	MW(WORD_STRONG :=  MesBlock3_Temp[1  ],	WORD_WEAK := MesBlock3_Temp[2  ], SIZE := 2, FIX := 3, SIGNED := 1, VAR_OUT	:= MesDataExd.MesData.MesIdc);
	MW(WORD_STRONG :=  MesBlock3_Temp[3  ],	WORD_WEAK := MesBlock3_Temp[4  ], SIZE := 2, FIX := 2, SIGNED := 1, VAR_OUT	:= MesDataExd.MesData.MesUdc);
	MW(WORD_STRONG :=  MesBlock3_Temp[5  ],	WORD_WEAK := MesBlock3_Temp[6  ], SIZE := 2, FIX := 0, SIGNED := 1, VAR_OUT	:= MesDataExd.MesData.MesPdc);
	MW(WORD_STRONG :=  MesBlock3_Temp[7  ],	WORD_WEAK := MesBlock3_Temp[8  ], SIZE := 2, FIX := 0, SIGNED := 1, VAR_OUT	:= MesDataExd.MesData.MesP);
	MW(WORD_STRONG :=  MesBlock3_Temp[21 ],	WORD_WEAK := MesBlock3_Temp[22 ], SIZE := 2, FIX := 2, SIGNED := 0, VAR_OUT	:= MesDataExd.MesU12);
	MW(WORD_STRONG :=  MesBlock3_Temp[23 ],	WORD_WEAK := MesBlock3_Temp[24 ], SIZE := 2, FIX := 2, SIGNED := 0, VAR_OUT	:= MesDataExd.MesU23);
	MW(WORD_STRONG :=  MesBlock3_Temp[25 ],	WORD_WEAK := MesBlock3_Temp[26 ], SIZE := 2, FIX := 2, SIGNED := 0, VAR_OUT	:= MesDataExd.MesU31);
	MW(WORD_STRONG :=  MesBlock3_Temp[27 ],	WORD_WEAK := MesBlock3_Temp[28 ], SIZE := 2, FIX := 3, SIGNED := 0, VAR_OUT	:= MesDataExd.MesData.MesI);
	MW(WORD_STRONG :=  MesBlock3_Temp[29 ],	WORD_WEAK := MesBlock3_Temp[30 ], SIZE := 2, FIX := 3, SIGNED := 0, VAR_OUT	:= MesDataExd.MesI1);
	MW(WORD_STRONG :=  MesBlock3_Temp[31 ],	WORD_WEAK := MesBlock3_Temp[32 ], SIZE := 2, FIX := 3, SIGNED := 0, VAR_OUT	:= MesDataExd.MesI2);
	MW(WORD_STRONG :=  MesBlock3_Temp[33 ],	WORD_WEAK := MesBlock3_Temp[34 ], SIZE := 2, FIX := 3, SIGNED := 0, VAR_OUT	:= MesDataExd.MesI3);
	MW(WORD_STRONG :=  MesBlock3_Temp[35 ],	WORD_WEAK := MesBlock3_Temp[36 ], SIZE := 2, FIX := 2, SIGNED := 0, VAR_OUT	:= MesDataExd.MesData.MesFreq);
	MW(WORD_STRONG :=  MesBlock3_Temp[37 ],	WORD_WEAK := MesBlock3_Temp[38 ], SIZE := 2, FIX := 2, SIGNED := 1, VAR_OUT	:= MesDataExd.MesData.MesQ);
	MW(WORD_STRONG :=  MesBlock3_Temp[53 ],	WORD_WEAK := MesBlock3_Temp[54 ], SIZE := 2, FIX := 2, SIGNED := 0, VAR_OUT	:= MesDataExd.MesData.MesCosPhi);
	MW(WORD_STRONG :=  MesBlock3_Temp[55 ],	WORD_WEAK := MesBlock3_Temp[56 ], SIZE := 2, FIX := 0, SIGNED := 0, VAR_OUT	:= MesDataExd.MesTypeCosPhi);
	MW(WORD_STRONG :=  MesBlock3_Temp[57 ],	WORD_WEAK := MesBlock3_Temp[58 ], SIZE := 2, FIX := 0, SIGNED := 0, VAR_OUT	:= MesDataExd.MesQMode);
	MW(WORD_STRONG :=  MesBlock3_Temp[59 ],	WORD_WEAK := MesBlock3_Temp[60 ], SIZE := 2, FIX := 0, SIGNED := 1, VAR_OUT	:= MesDataExd.MesSetptQ);
	MW(WORD_STRONG :=  MesBlock3_Temp[61 ],	WORD_WEAK := MesBlock3_Temp[62 ], SIZE := 2, FIX := 1, SIGNED := 1, VAR_OUT	:= MesDataExd.MesSetptQ_Pct);
	MW(WORD_STRONG :=  MesBlock3_Temp[63 ],	WORD_WEAK := MesBlock3_Temp[64 ], SIZE := 2, FIX := 2, SIGNED := 1, VAR_OUT	:= MesDataExd.MesSetptCosPhi);
	MW(WORD_STRONG :=  MesBlock3_Temp[65 ],	WORD_WEAK := MesBlock3_Temp[66 ], SIZE := 2, FIX := 0, SIGNED := 0, VAR_OUT	:= MesDataExd.MesSetptType_CosPhi);
	MW(WORD_STRONG :=  MesBlock3_Temp[67 ],	WORD_WEAK := MesBlock3_Temp[68 ], SIZE := 2, FIX := 0, SIGNED := 0, VAR_OUT	:= MesDataExd.MesPMode);
	MW(WORD_STRONG :=  MesBlock3_Temp[69 ],	WORD_WEAK := MesBlock3_Temp[70 ], SIZE := 2, FIX := 0, SIGNED := 0, VAR_OUT	:= MesDataExd.MesPSetpt);
	MW(WORD_STRONG :=  MesBlock3_Temp[71 ],	WORD_WEAK := MesBlock3_Temp[72 ], SIZE := 2, FIX := 0, SIGNED := 0, VAR_OUT	:= MesDataExd.MesPSetptPct);
	MW(WORD_STRONG :=  MesBlock3_Temp[73 ],	WORD_WEAK := MesBlock3_Temp[74 ], SIZE := 2, FIX := 2, SIGNED := 0, VAR_OUT	:= MesDataExd.MesData.MesV);
	
	MW(WORD_STRONG :=  MesBlock4_Temp[1  ],	WORD_WEAK := MesBlock4_Temp[2  ], SIZE := 2, FIX := 1, SIGNED := 1, VAR_OUT	:= MesDataExd.MesTmpHs);
	MW(WORD_STRONG :=  MesBlock4_Temp[5  ],	WORD_WEAK := MesBlock4_Temp[6  ], SIZE := 2, FIX := 1, SIGNED := 1, VAR_OUT	:= MesDataExd.MesTmpCab1);
	MW(WORD_STRONG :=  MesBlock4_Temp[9  ],	WORD_WEAK := MesBlock4_Temp[10 ], SIZE := 2, FIX := 1, SIGNED := 1, VAR_OUT	:= MesDataExd.MesTmpCab3);
	MW(WORD_STRONG :=  MesBlock4_Temp[17 ],	WORD_WEAK := MesBlock4_Temp[18 ], SIZE := 2, FIX := 1, SIGNED := 1, VAR_OUT	:= MesDataExd.MesTmpExt);
	MW(WORD_STRONG :=  MesBlock4_Temp[37 ],	WORD_WEAK := MesBlock4_Temp[38 ], SIZE := 2, FIX := 1, SIGNED := 1, VAR_OUT	:= MesDataExd.MesTmpCol);
			                                                                                                                          

	MW(WORD_STRONG :=  MesBlock5_Temp[1  ],	WORD_WEAK := MesBlock5_Temp[2  ], SIZE := 2, FIX := 0, SIGNED := 0, VAR_OUT	:= MesDataExd.MesGHI);
	MW(WORD_STRONG :=  MesBlock5_Temp[25 ],	WORD_WEAK := MesBlock5_Temp[26 ], SIZE := 2, FIX := 0, SIGNED := 0, VAR_OUT	:= MesDataExd.MesInCur1);
	MW(WORD_STRONG :=  MesBlock5_Temp[27 ],	WORD_WEAK := MesBlock5_Temp[28 ], SIZE := 2, FIX := 0, SIGNED := 0, VAR_OUT	:= MesDataExd.MesInCur2);

	
	MW(WORD_STRONG :=  MesBlock6_Temp[1  ],	WORD_WEAK := MesBlock6_Temp[2  ], SIZE := 2, FIX := 0, SIGNED := 0, VAR_OUT	:= PosInterm);
	MesDataExd.MesOpStateOn := SEL(PosInterm = 381,SEL(PosInterm=569,FALSE, TRUE), FALSE);
	MW(WORD_STRONG :=  MesBlock6_Temp[12 ],	WORD_WEAK := MesBlock6_Temp[13 ], SIZE := 2, FIX := 0, SIGNED := 0, VAR_OUT	:= PosInterm);
	MesDataExd.MesbRIsoOn := SEL(PosInterm=303,SEL(PosInterm=308,FALSE, TRUE), FALSE);
	IdcTotal := 0;


	IF FB_ModbusRead[7].OUT_NbRead > 0 THEN 
		
		MW(WORD_STRONG :=  MesBlock7_Temp[1 ],	WORD_WEAK := MesBlock7_Temp[2], SIZE := 2, FIX := 3, SIGNED := 1, VAR_OUT	:= MesDataExd.BJMonitor[ID_SSM].AX_STR[1].MesData.MesIdc);
		MW(WORD_STRONG :=  MesBlock7_Temp[3 ],	WORD_WEAK := MesBlock7_Temp[4], SIZE := 2, FIX := 3, SIGNED := 1, VAR_OUT	:= MesDataExd.BJMonitor[ID_SSM].AX_STR[2].MesData.MesIdc);
		MW(WORD_STRONG :=  MesBlock7_Temp[5 ],	WORD_WEAK := MesBlock7_Temp[6 ], SIZE := 2, FIX := 3, SIGNED := 1, VAR_OUT	:= MesDataExd.BJMonitor[ID_SSM].AX_STR[3].MesData.MesIdc);
		MW(WORD_STRONG :=  MesBlock7_Temp[7 ],	WORD_WEAK := MesBlock7_Temp[8 ], SIZE := 2, FIX := 3, SIGNED := 1, VAR_OUT	:= MesDataExd.BJMonitor[ID_SSM].AX_STR[4].MesData.MesIdc);
		MW(WORD_STRONG :=  MesBlock7_Temp[9 ],	WORD_WEAK := MesBlock7_Temp[10], SIZE := 2, FIX := 3, SIGNED := 1, VAR_OUT	:= MesDataExd.BJMonitor[ID_SSM].AX_STR[5].MesData.MesIdc);
		MW(WORD_STRONG :=  MesBlock7_Temp[11],	WORD_WEAK := MesBlock7_Temp[12], SIZE := 2, FIX := 3, SIGNED := 1, VAR_OUT	:= MesDataExd.BJMonitor[ID_SSM].AX_STR[6].MesData.MesIdc);
		MW(WORD_STRONG :=  MesBlock7_Temp[13],	WORD_WEAK := MesBlock7_Temp[14], SIZE := 2, FIX := 3, SIGNED := 1, VAR_OUT	:= MesDataExd.BJMonitor[ID_SSM].AX_STR[7].MesData.MesIdc);
		MW(WORD_STRONG :=  MesBlock7_Temp[15],	WORD_WEAK := MesBlock7_Temp[16], SIZE := 2, FIX := 3, SIGNED := 1, VAR_OUT	:= MesDataExd.BJMonitor[ID_SSM].AX_STR[8].MesData.MesIdc);	
	
			
		//	MW(WORD_STRONG :=  MesBlock8_Temp[1],	WORD_WEAK := MesBlock8_Temp[2 ], SIZE := 2, FIX := 2, SIGNED := 0, VAR_OUT	:= PosInterm);
		//MesDataExd.BJMonitor.MesID_SignalContact1 := SEL(PosInterm=303,SEL(PosInterm=308,FALSE, TRUE), FALSE);
		MesDataExd.BJMonitor[ID_SSM].MesID_SignalContact1 := MesBlock8_Temp[1] ; 
		//	MW(WORD_STRONG :=  MesBlock8_Temp[3],	WORD_WEAK := MesBlock8_Temp[4 ], SIZE := 2, FIX := 2, SIGNED := 0, VAR_OUT	:= PosInterm);
		//MesDataExd.BJMonitor.MesID_SignalContact2 := SEL(PosInterm=303,SEL(PosInterm=308,FALSE, TRUE), FALSE);
		MesDataExd.BJMonitor[ID_SSM].MesID_SignalContact2 := MesBlock8_Temp[3] ; 
			

		ID_SSM := ID_SSM +1 MOD 7 ; 
		IF ID_SSM = 0 THEN 
			ID_SSM := 1 ; 
		END_IF
	END_IF




	MesDataExd.MesData.MesP := MesDataExd.MesData.MesP/1000;
	MesDataExd.MesData.MesPdc := MesDataExd.MesData.MesPdc/1000;
	MesDataExd.MesData.MesQ := MesDataExd.MesData.MesQ/1000;
	MesDataExd.MesPSetpt := MesDataExd.MesPSetpt / 1000;
	MesDataExd.MesSetptQ := MesDataExd.MesSetptQ / 1000;

	
	
END_IF
	
	
// Update value 
MesDataExd.Mesdata.ParamPn		:= ParamPn ; 
MesDataExd.Mesdata.ParamQn		:= ParamQn ; 
	


FOR KK := 1 TO CstNbSB_INV_G DO 
	MesDataExd.BJMonitor[KK].MesClosed_DCSwitch := IN_MesClosed_BJ_IO[KK] ; 
END_FOR
END_METHOD

METHOD M_StartStop 
VAR_INPUT
END_VAR
VAR
	KK : UINT;
	AX_ADR_MB			: WORD := 40009;
	AX_QTY_MB			: ARRAY[1..2] OF BYTE := [2, 2];
	MotStart			: WORD := 569;
	MotStop				: WORD := 381;
	
END_VAR
SUPER^.M_StartStop() ; 
FB_ModbusWrite[3](WriteCmd := FALSE);

//Read the setpoints
	// Evaluate the cmd given 

	StartStop_RTrig(CLK:=CalCP_CMD_StartStop);
	StartStop_RTrigIO(CLK:=CalCP_CMD_StartStopIO);
	
//	IF StartStop_RTrig.Q THEN
		IF RS_StartStop.Q1 THEN
			MesBlockWrite3_Temp[1] := 0;
			MesBlockWrite3_Temp[2] := MotStart;
		ELSE 
			MesBlockWrite3_Temp[1] := 0;
			MesBlockWrite3_Temp[2] := MotStop;
		END_IF
//	END_IF
	
//	IF StartStop_RTrigIO.Q THEN
//		IF Cmd_SwitchOff THEN
//			Cmd_SwitchOff		:= 0;
//		ELSIF NOT Cmd_SwitchOff THEN
//			Cmd_SwitchOff		:= 1;
//		END_IF
//	END_IF
OUT_Cmd_SwitchOff_IO	:= CalCP_CMD_StartStopIO	;
	

MesDataExd.Mesdata.OUT_CmdStart := RS_StartStop.Q1 ;
MesDataExd.Mesdata.OUT_CmdStop := NOT RS_StartStop.Q1 ;

	
	FB_ModbusWrite[3]
	(
		pSrcAddr := ADR (MesBlockWrite3_Temp),
		sIPAddr := ParamIPAddress,
		tTimeout := ParamTimeout,
		nMBAddr := AX_ADR_MB,
		nTCPport := ParamTCPPort,
		cbLength := SIZEOF(MesBlockWrite3_Temp),
		nQuantity := 2,
		nUnitID := 3,
		WriteCmd := CalCP_CMD_StartStop AND MesDataExd.mesData.MesCP_Write ,
		Reset := CmdClearFault_G,
		ErrorId => AX_ModbusWriteAlarmId[3],
		ModbusWriteAlarm => AX_ModbusWriteAlarm[3]
	);


SUPER^.M_Curtail() ;
END_METHOD

METHOD M_StateManager
//////////////////
// Detect which is the state of the inverter. IF loss of communication MesState =0 , the last inverter state is kept .  
/////////////////

VAR 
	// Method local variables (reinitialized at each cycle) 

	
END_VAR
// 0 = Stopped, 1 = MPPT, 2 = Sleeping, 3 = Starting, 4 = Throttled, 5 = Shutting down, 6 = Fault, 7 = Standby

MesDataExd.Mesdata.MesState 			:= 0  ; 

IF MesDataExd.mesData.MesState_Inv = 381 OR MesDataExd.mesData.MesState_Inv = 1455 THEN // IF INVERTER IS STOPPED 309 = Operation && 455 = warning
	MesDataExd.Mesdata.MesState.0 := 1;		// Stop
ELSIF MesDataExd.mesData.MesState_Inv = 295 THEN
	MesDataExd.Mesdata.MesState.1 := 1;
ELSIF MesDataExd.mesData.MesState_Inv = 1466 THEN // Wait 
	MesDataExd.Mesdata.MesState.7 := 1;
ELSIF MesDataExd.mesData.MesState_Inv = 1467 OR MesDataExd.mesData.MesState_Inv = 1468 OR MesDataExd.mesData.MesState_Inv = 1479 THEN
	MesDataExd.Mesdata.MesState.3 := 1;
ELSIF MesDataExd.mesData.MesState_Inv = 1469  THEN
	MesDataExd.Mesdata.MesState.5 := 1;
ELSIF MesDataExd.mesData.MesState_Inv = 1470  THEN
	MesDataExd.Mesdata.MesState.6 := 1;
ELSE 
	MesDataExd.Mesdata.MesState.0 := 1;
END_IF

//IF MesDataExd.Mesdata.OUT_SetptP < ParamPn AND MesDataExd.Mesdata.MesP > 0.95 * MesDataExd.Mesdata.OUT_SetptP THEN
//	MesDataExd.Mesdata.MesIDState.4 := 1;
//END_IF



SUPER^.M_StateManager() ;
END_METHOD

END_FUNCTION_BLOCK

// ---- 01_Equipement_Library/Inverter/FB_INV_SmaSCXXXXUP_US.TcPOU
FUNCTION_BLOCK FB_INV_SmaSCXXXXUP_US EXTENDS FB_INV_Base
// Reading through Webbox . Curtailement not possible through modbus . 
//

VAR_INPUT PERSISTENT
	ParamTcpPort				: UINT	:= 502 ;	(* Modbus TCP port*)
	//{attribute 'OPC.UA.DA' := '1'} 
	//ParamQn						: REAL ;		(* (kVAr) Nominal Reactive Power*)
	{attribute 'OPC.UA.DA' := '1'} 
	ParamIPAddress				: STRING; 			(* (NA)Config: IP Adress of PV INverter	*)
	{attribute 'OPC.UA.DA' := '1'} 
	ParamUnitID 				: BYTE := 3; 			(* (NA)   SMA Modbus Unit ID. *)
	ParamNumInv					: BYTE;             (* Inverter Index  *)
	ParamNbSB					: BYTE :=5 ; (* Number of String Box per inverter*)
	ParamNbSTR					: BYTE :=8 ; (* Number of String per string Box*)
	
//	ParamUnitID_STR				: ARRAY[1..CstNbSB_INV_G] OF BYTE ; (* Unit ID Arrray for each string box . *)
	
	ParamDelayReadSTR			: TIME := T#2S ; 			(* (s) Delay after inv data read , to read string values . 	*)

END_VAR

VAR_INPUT 
	// Parameters of the Object (instance specific) 
	       	MesDataExd					: INV_SmaSCXXXXUP_US;
	                                     	
END_VAR

VAR
		
	// M_ALARMMNGMT VARIABLES //
	
	// M_READ VARIABLES//
		//MesDataCC_Read				:  INV_CC;	
		//MesDataCC_Cmd				:  INV_CC;
		
	
		FB_ModbusRead	          	: ARRAY[1..6] OF FB_ModbusReadInputRegs; 	            // (NA) FB for Modbus Reading
		FB_ModbusWrite				: ARRAY[1..3] OF FB_ModbusWrite;
		AX_ModbusReadAlarm			: ARRAY[1..6] OF BOOL;
		AX_ModbusReadAlarmId		: ARRAY[1..6] OF UDINT;		
		AX_ModbusWriteAlarm			: ARRAY[1..2] OF BOOL;
		AX_ModbusWriteAlarmId		: ARRAY[1..2] OF UDINT;
	

		
		MesBlock_Temp_1 				: ARRAY [1..125] OF WORD ; 		// (NA) Temporary Block with multiple modbus reading (Caution : Double Word variables)
		MesBlock_Temp_2 				: ARRAY [1..125] OF WORD ; 		// (NA) Temporary Block with multiple modbus reading (Caution : Double Word variables)
		MesBlock_Temp_3 				: ARRAY [1..125] OF WORD ; 		// (NA) Temporary Block with multiple modbus reading (Caution : Double Word variables)
		MesBlock_Temp_4 				: ARRAY [1..20] OF WORD ; 		// (NA) Temporary Block with multiple modbus reading (Caution : Double Word variables)
		MesBlock_Temp_5 				: ARRAY [1..20] OF WORD ; 		// (NA) Temporary Block with multiple modbus reading (Caution : Double Word variables)
		MesBlock_Temp_6				: ARRAY [1..20] OF WORD ;		// (NA) Temporary block with both start commands for each inverter


		MesBlockWrite3_Temp			: ARRAY [1..2] OF WORD ;
		
		TON_ReadSTR					: TON ; // Manage time delay fro reading string values. 
		
	// M_STARTSTOP//
	
		
	
	//  CUrtail 
	
		InvSetptP_temp		: WORD;
		InvSetptQ_temp		: WORD;
		
		MesBlockWrite1_Temp : WORD ; 
		MesBlockWrite2_Temp : WORD ; 
		
		
	// M_CP
		CalCP_CMD_StartStop			: BOOL ; 		  // Write command start;
	
	// M_STATEMANAGER//
	
	//M_EXECUTE VARIABLES //
	//	bInit						: BOOL ;
	//EMULATOR VARIABLES //
		
END_VAR

METHOD M_AlarmManagement
//////////////////
// Manages IntelliGen Alarms
/////////////////

VAR 
	// Method local variables (reinitialized at each cycle) 
	FB_AlarmCodeManager : FB_AlarmCodeManager ; 
	KK				: BYTE;		// For Loop 
	bComError		: BOOL := TRUE;
	bComWarning 	: BOOL;

END_VAR
FOR KK := 1 TO 4 DO
	bCOmError := bCOmError AND FB_ModbusRead[KK].ModbusReadAlarm;
	bComWarning := bComWarning OR FB_ModbusRead[KK].ModbusReadAlarm;
END_FOR
bComError := bComError AND FB_ModbusWrite[1].ModbusWriteAlarm ;
bComWarning := bComError OR FB_ModbusWrite[1].ModbusWriteAlarm  ;

TON_ComAlarm(IN := bComError, PT := T#30S , Q=> MesDataExd.MesData.MesAlarmCom);
TON_ComWarning(IN := bComWarning, PT := T#30S);



// ALARM CODE //
	FB_AlarmCodeManager(
		bAlarm1			:= MesDataExd.MesData.MesState_Inv  = 1392	, 	//Inverter in error  #Equipment
		bAlarm2			:= MesDataExd.MesData.MesState_Inv = 381,		// INV in stopped mode  #Equipment
		bAlarm3			:= MesDataExd.MesID_ErrorState = 1392 , 		// INV error synthesis #Equipment 
		bAlarm4			:= MesDataExd.Mesdata.MesOpened_Ac , 			// AC Switch is opened #Equipment
		bAlarm5			:= MesDataExd.Mesdata.MesOpened_Dc, 			// All DC switch are opened 
		bAlarm6			:= FALSE , //
		bAlarm7			:= FALSE , //
		bAlarm8			:= FALSE,						// 
		bAlarm9			:= FALSE	,					//
		bAlarm10		:= FALSE , 							// 
		bAlarm11		:= FALSE,								// 
		bAlarm12		:= FALSE,								// 
		bAlarm13		:= FALSE,  								//
		bAlarm14		:= FALSE,								// 
		bAlarm15		:= MesDataExd.MesData.MesAlarmCom, 						// No communication frames for the past 30 seconds #COM
		wAlarmCode		=> mesdataExd.MesData.MesAlarmCode);

// WARNING CODE //
	FB_AlarmCodeManager(
 		bAlarm1			:= FALSE, 													// 
		bAlarm2			:= FALSE,
		bAlarm3			:= NOT MesDataExd.MesData.MesCP_Read, 	  							// Reading has been disabled
		bAlarm4			:= FALSE,															// 
		bAlarm5			:= NOT MesDataExd.MesData.MesCP_Write,								// Writing has been disabled			
		bAlarm6			:= MesDataExd.MesID_DC1State = 311 OR MesDataExd.MesID_DC2State = 311 OR MesDataExd.MesID_DC3State = 311, // At least one DC switch is opened 								// 
		bAlarm7			:= FALSE , //
		bAlarm8			:= FALSE, 															//
		bAlarm9			:= FALSE, 								// 
		bAlarm10		:= NOT RS_StartStop_Local.Q1,                  						// Local Stop Command, 
		bAlarm11		:= FALSE, //
		bAlarm12		:= FALSE, //
		bAlarm13		:= FALSE, //
		bAlarm14		:= FALSE, //
		bAlarm15		:= TON_ComWarning.Q, 												//One or more than error, communication frames for the past 30 seconds #COM
		wAlarmCode		=> MesDataExd.mesdata.MesWarningCode);	

// EVENT CODE //
	FB_AlarmCodeManager(
		bAlarm1			:= MesDataExd.MesData.MesState_Inv = 1787, 								// Inverter status : Init  #Equipment
		bAlarm2			:= MesDataExd.MesData.MesState_Inv = 3522,								// Inverter status : Update  #Equipment
		bAlarm3			:= MesDataExd.MesData.MesState_Inv = 3523,								// Inverter status : Reset  #Equipment
		bAlarm4			:= MesDataExd.MesData.MesState_Inv = 1394,								// Inverter status : WaitAC  #Equipment
		bAlarm5			:= MesDataExd.MesData.MesState_Inv = 3524,								// Inverter status : ConnectAC  #Equipment
		bAlarm6			:= MesDataExd.MesData.MesState_Inv = 1393,								// Inverter status : WaitDC  #Equipment
		bAlarm7			:= NOT RS_StartStop.Q1, 				// Stop command for INV1
		bAlarm8			:= MesDataExd.MesData.MesState_Inv = 3525,								// Inverter status : ConnectDC  #Equipment
		bAlarm9			:= MesDataExd.MesData.MesState_Inv = 3526,								// Inverter status : GridFeed  #Equipment
		bAlarm10		:= MesDataExd.MesData.MesState_Inv = 3527,								// Inverter status : FRT  #Equipment
		bAlarm11		:= MesDataExd.MesData.MesState_Inv = 3528,								// Inverter status : Standby  #Equipment
		bAlarm12		:= MesDataExd.MesData.MesState_Inv = 3529,								// Inverter status : QonDemand  #Equipment
		bAlarm13		:= MesDataExd.MesData.MesState_Inv = 3530,								// Inverter status : RampDown   #Equipment
		bAlarm14		:= MesDataExd.MesData.MesState_Inv = 1469,								// Inverter status : ShutDown  #Equipment
		bAlarm15		:= MesDataExd.MesData.MesState_Inv = 375,								// Inverter status : Selftest  #Equipment
		wAlarmCode		=> mesdataExd.MesData.MesEventCode);

FB_AlarmCodeManager(
		bAlarm1			:= MesDataExd.MesID_Derating = 21585, 								// Inverter Derating : Stk.DcAmpLim  #Equipment
		bAlarm2			:= MesDataExd.MesID_Derating = 21586,								// Inverter Derating : Frt  #Equipment
		bAlarm3			:= MesDataExd.MesID_Derating = 21587,								// Inverter Derating : AmpGra  #Equipment
		bAlarm4			:= MesDataExd.MesID_Derating = 21588,								// Inverter Derating : AMax  #Equipment
		bAlarm5			:= MesDataExd.MesID_Derating = 21589,								// Inverter Derating : VAMax  #Equipment
		bAlarm6			:= MesDataExd.MesID_Derating = 21590,								// Inverter Derating : WCtlLoHz  #Equipment
		bAlarm7			:= MesDataExd.MesID_Derating = 21591,								// Inverter Derating : WCtlHz  #Equipment
		bAlarm8			:= MesDataExd.MesID_Derating = 21592,								// Inverter Derating : WGraRecon  #Equipment
		bAlarm9			:= MesDataExd.MesID_Derating = 21593,								// Inverter Derating : WGra  #Equipment
		bAlarm10		:= MesDataExd.MesID_Derating = 21594,								// Inverter Derating : WMax  #Equipment
		bAlarm11		:= MesDataExd.MesID_Derating = 21595,								// Inverter Derating : WMaxExt  #Equipment
		bAlarm12		:= MesDataExd.MesID_Derating = 21596,								// Inverter Derating : VecLen  #Equipment
		bAlarm13		:= MesDataExd.MesID_Derating = 21599,								// Inverter Derating : WGraStr   #Equipment
		bAlarm14		:= MesDataExd.MesID_Derating = 21601,								// Inverter Derating : WCtlVol  #Equipment
		bAlarm15		:= MesDataExd.MesID_Derating = 21602,								// Inverter Derating : Mvps.WRvLim  #Equipment
		wAlarmCode		=> mesdataExd.MesStatus_Derating);

FB_AlarmCodeManager(
		bAlarm1			:= MesDataExd.MesID_Derating = 21651, 								// Inverter Derating : VArPrio  #Equipment
		bAlarm2			:= FALSE,
		bAlarm3			:= FALSE,
		bAlarm4			:= FALSE,
		bAlarm5			:= FALSE,
		bAlarm6			:= FALSE,
		bAlarm7			:= FALSE,
		bAlarm8			:= FALSE,
		bAlarm9			:= FALSE,
		bAlarm10		:= FALSE,
		bAlarm11		:= FALSE,
		bAlarm12		:= FALSE,
		bAlarm13		:= FALSE,
		bAlarm14		:= FALSE,
		bAlarm15		:= FALSE,
		wAlarmCode		=> mesdataExd.MesStatus_Derating1);


	FB_AlarmCodeManager(
		bAlarm1			:= MesDataExd.MesID_Off = 21604, 								// Off Reason : Error: Critical Error, ProErr active  #Equipment
		bAlarm2			:= MesDataExd.MesID_Off = 21605,								// Off Reason : Error  #Equipment
		bAlarm3			:= MesDataExd.MesID_Off = 21606,								// Off Reason : Stop: Key Switch  #Equipment
		bAlarm4			:= MesDataExd.MesID_Off = 21607,								// Off Reason : Stop: Parameter InvOpmod  #Equipment
		bAlarm5			:= MesDataExd.MesID_Off = 21608,								// Off Reason : Stop: Stop External X440:3  #Equipment
		bAlarm6			:= MesDataExd.MesID_Off = 21609,								// Off Reason : Stop: Scada or PPC, Modbus  #Equipment
		bAlarm7			:= MesDataExd.MesID_Off = 21610,								// Off Reason : Stop: unspecified  #Equipment
		bAlarm8			:= MesDataExd.MesID_Off = 21612,								// Off Reason : Standby: Scada or PPC, Modbus
		bAlarm9			:= MesDataExd.MesID_Off = 21613,								// Off Reason : Standby: AC Synchronization  #Equipment     
		bAlarm10		:= MesDataExd.MesID_Off = 21614,								// Off Reason : Standby: Low DC Power  #Equipment           
		bAlarm11		:= MesDataExd.MesID_Off = 21615,								// Off Reason : Standby: External Grid Error  #Equipment    
		bAlarm12		:= MesDataExd.MesID_Off = 21616,								// Off Reason : Standby: Power Monitoring Module  #Equipment
		bAlarm13		:= MesDataExd.MesID_Off = 21617,								// Off Reason : Standby: Parameter RemRdy   #Equipment      
		bAlarm14		:= MesDataExd.MesID_Off = 21618,								// Off Reason : Standby External X440:7  #Equipment         
		bAlarm15		:= MesDataExd.MesID_Off = 21619,								// Off Reason : Standby: unspecified  #Equipment            
		wAlarmCode		=> mesdataExd.MesStatus_Off);


	FB_AlarmCodeManager(
		bAlarm1			:= MesDataExd.MesID_Off = 21620, 								// Off Reason : WaitAc  #Equipment
		bAlarm2			:= MesDataExd.MesID_Off = 21621,								// Off Reason : WaitDc: DC Voltage  #Equipment
		bAlarm3			:= MesDataExd.MesID_Off = 21622,								// Off Reason : WaitDc: Bender  #Equipment
		bAlarm4			:= MesDataExd.MesID_Off = 21623,								// Off Reason : WaitDc: DC precharge waiting period  #Equipment
		bAlarm5			:= MesDataExd.MesID_Off = 21624,								// Off Reason : Selftest active  #Equipment
		bAlarm6			:= MesDataExd.MesID_Off = 21625,								// Off Reason : IO Test active  #Equipment
		bAlarm7			:= MesDataExd.MesID_Off = 21626,								// Off Reason : Low Power Set Point  #Equipment
		bAlarm8			:= FALSE,
		bAlarm9			:= FALSE,
		bAlarm10		:= FALSE,
		bAlarm11		:= FALSE,
		bAlarm12		:= FALSE,
		bAlarm13		:= FALSE,
		bAlarm14		:= FALSE,
		bAlarm15		:= MesDataExd.MesID_Off = 21623,							// Inverter status : Selftest  #Equipment
		wAlarmCode		=> mesdataExd.MesStatus_Off1);
END_METHOD

METHOD M_CP
//////////////////
//  Emulator
/////////////////

VAR 
	// Method local variables (reinitialized at each cycle) 
	MesOpState : BOOL;
END_VAR


SUPER^.M_CP() ; 




Trig_Cmd_Read(CLK:=IN_CmdToggleRead);
Trig_Cmd_Write(CLK:=IN_CmdToggleWrite);
	
IF Trig_Cmd_Read.Q THEN
	IN_CmdToggleRead := FALSE;
	MesDataExd.MesData.MesCP_Read := NOT MesDataExd.MesData.MesCP_Read;
END_IF


IF Trig_Cmd_Write.Q THEN
	IN_CmdToggleWrite := FALSE;
	MesDataExd.MesData.MesCP_Write := NOT MesDataExd.MesData.MesCP_Write;
END_IF
END_METHOD

{attribute 'object_name' := 'M_Curtail'}
METHOD M_Curtail
//////////////////
// Write Curtail Command through modbus to PV inverters.  
//////////////////
VAR 
	// Method local variables (reinitialized at each cycle) 

	AX_ADR_MB			: WORD := 40022;
	AX_QTY_MB			: BYTE := 2;
	AX_UnitID_MB		: BYTE := 2;
	
	KK: INT;
END_VAR
SUPER^.M_Curtail() ; 
// MODBUS VARIABLE FORMATING //
FB_ModbusWrite[1](WriteCmd := FALSE);

MesDataExd.MesData.OUT_SetptPLimit :=  IN_SetptPlimit ; 
MesDataExd.MesData.OUT_SetptQ :=  IN_SetptQ ; 

InvSetptP_temp	:= REAL_TO_WORD(IN_SetptPlimit*100 / ParamPn)*100;
InvSetptQ_temp	:= REAL_TO_WORD(IN_SetptQ*100 / ParamQn)*100;

		
IF A1_PP.ParamTanPhiCtrl  OR A1_SUBMV.A1_GRID.MesDataExd.OUT_CmdQReg	THEN
	MesBlockWrite1_Temp	:= InvSetptP_temp;	
	MesBlockWrite2_Temp	:= InvSetptQ_temp;
ELSE
	MesBlockWrite1_Temp:= InvSetptP_temp;
	MesBlockWrite2_Temp:= 0;
	
 
END_IF

FB_ModbusWrite[1]
(
	pSrcAddr := ADR (MesBlockWrite1_Temp),
	sIPAddr := ParamIPAddress,
	tTimeout := ParamTimeout,
	nMBAddr := 40023,
	nTCPport := ParamTCPPort,
	cbLength := SIZEOF(MesBlockWrite1_Temp),
	nQuantity := 1,
	nUnitID := 2,
	WriteCmd := ClockWrite AND MesDataExd.Mesdata.MesCP_Write  ,
	Reset := CmdClearFault_G OR IN_CmdReset_L,
	ErrorId => AX_ModbusWriteAlarmId[1],
	ModbusWriteAlarm => AX_ModbusWriteAlarm[1]
);

FB_ModbusWrite[2]
(
	pSrcAddr := ADR (MesBlockWrite2_Temp),
	sIPAddr := ParamIPAddress,
	tTimeout := ParamTimeout,
	nMBAddr := 40022,
	nTCPport := ParamTCPPort,
	cbLength := SIZEOF(MesBlockWrite2_Temp),
	nQuantity := 1,
	nUnitID := 2,
	WriteCmd := ClockWrite AND MesDataExd.Mesdata.MesCP_Write  ,
	Reset := CmdClearFault_G OR IN_CmdReset_L,
	ErrorId => AX_ModbusWriteAlarmId[2],
	ModbusWriteAlarm => AX_ModbusWriteAlarm[2]
);
END_METHOD

METHOD M_Execute
//////////////////
//  Method Calls 
/////////////////

VAR 
	// Method local variables (reinitialized at each cycle) 

END_VAR
IF bInit THEN
	M_Init();
END_IF


SUPER^.M_Execute() ;
END_METHOD

METHOD M_Init
VAR_INPUT
END_VAR

VAR

END_VAR
ParamPn := 4200;
ParamQn := 2520;
RS_StartStop_Local(SET:= TRUE ); 
RS_StartStop_Local(SET:= FALSE ); 
IN_SetptPlimit_Local := ParamPn ;
//Trig_Cmd_Read(CLK:=TRUE);
//Trig_Cmd_Write(CLK:=TRUE);
IN_CmdStart_Local := TRUE;
bInit := FALSE;
END_METHOD

{attribute 'object_name' := 'M_Read'}
METHOD M_Read
//////////
// Read Method for SMA : Modbus reading
//////////
VAR
	// Method local variables (reinitialized at each cycle) 
	
	MW					: FB_MergeWordsToDint;
	MW_U				: FB_MergeWordsToUint;
	AX_QTY_MB			: ARRAY[1..6] OF WORD := [124,	103, 	10, 	10];
	AX_ADR_MB			: ARRAY[1..6] OF WORD := [0,	124, 	55, 	55];
	

	kk: UINT;

	JJ: UINT;
END_VAR
TON_ReadSTR(IN:= ClockRead, PT:= ParamDelayReadSTR) ; 

IF MesDataExd.MesData.MesCP_Read THEN		


// MODBUS REQUEST//
	//Electrical Measurements + Ground Measurements
	FB_ModbusRead[1]
	(
		nTCPPort	:= ParamTcpPort,
		ClockRead:= MesDataExd.MesData.MesCP_Read AND ClockRead, 
		Reset:= CmdClearFault_G OR IN_CmdReset_L,
		sIPAddr:=ParamIPAddress ,
		nUnitID:= ParamUnitID, 
		tTimeout:= ParamTimeout,
		nQuantity		:= AX_QTY_MB[1] , 
		nMBAddr			:= AX_ADR_MB[1] , 
		cbLength		:= SIZEOF(MesBlock_Temp_1) , 
		pDestAddr		:= ADR(MesBlock_Temp_1) , 
		ModbusReadAlarm	=>AX_ModbusReadAlarm[1] , 
		ErrorId			=> AX_ModbusReadAlarmId[1]
	);
	
	//Production Measurements
	FB_ModbusRead[2]
	(
		nTCPPort	:= ParamTcpPort,
		ClockRead:= MesDataExd.MesData.MesCP_Read AND ClockRead, 
		Reset:= CmdClearFault_G OR IN_CmdReset_L,
		sIPAddr:=ParamIPAddress , 
		nUnitID:= ParamUnitID, 
		tTimeout:= ParamTimeout,
		nQuantity		:= AX_QTY_MB[2] , 
		nMBAddr			:= AX_ADR_MB[2] , 
		cbLength		:= SIZEOF(MesBlock_Temp_2) , 
		pDestAddr		:= ADR(MesBlock_Temp_2) , 
		ModbusReadAlarm	=>AX_ModbusReadAlarm[2] , 
		ErrorId			=> AX_ModbusReadAlarmId[2]
	);
	
	(*
	FB_ModbusRead[3]
	(
		nTCPPort	:= ParamTcpPort,
		ClockRead:= mesdata.MesCP_Read AND ClockRead, 
		Reset:= CmdClearFault_G OR IN_CmdReset_L,
		sIPAddr:=ParamIPAddress , 
		nUnitID:= 32, 
		tTimeout:= ParamTimeout,
		nQuantity		:= AX_QTY_MB[3] , 
		nMBAddr			:= AX_ADR_MB[3] , 
		cbLength		:= SIZEOF(MesBlock_Temp_3) , 
		pDestAddr		:= ADR(MesBlock_Temp_3) , 
		ModbusReadAlarm	=>AX_ModbusReadAlarm[3] , 
		ErrorId			=> AX_ModbusReadAlarmId[3]
	);	
	
	FB_ModbusRead[4]
	(
		nTCPPort	:= ParamTcpPort,
		ClockRead:= mesdata.MesCP_Read AND ClockRead, 
		Reset:= CmdClearFault_G OR IN_CmdReset_L,
		sIPAddr:=ParamIPAddress , 
		nUnitID:= 33, 
		tTimeout:= ParamTimeout,
		nQuantity		:= AX_QTY_MB[4] , 
		nMBAddr			:= AX_ADR_MB[4] , 
		cbLength		:= SIZEOF(MesBlock_Temp_4) , 
		pDestAddr		:= ADR(MesBlock_Temp_4) , 
		ModbusReadAlarm	=>AX_ModbusReadAlarm[4] , 
		ErrorId			=> AX_ModbusReadAlarmId[4]
	);		
	*)
	
	
	
	// Bock 1 
		MW(WORD_STRONG:= MesBlock_Temp_1[ 1], Word_WEAK:= MesBlock_Temp_1[2], SIGNED:=TRUE, FIX:=1 , SIZE:=2, VAR_OUT:=MesDataExd.MesData.MesUdc);
		MW(WORD_STRONG:= MesBlock_Temp_1[ 3], Word_WEAK:= MesBlock_Temp_1[4], SIGNED:=TRUE, FIX:=0 , SIZE:=2, VAR_OUT:=MesDataExd.MesIdc_Group1);
		MW(WORD_STRONG:= MesBlock_Temp_1[ 5], Word_WEAK:= MesBlock_Temp_1[6], SIGNED:=TRUE, FIX:=0 , SIZE:=2, VAR_OUT:=MesDataExd.MesIdc_Group2);
		MW(WORD_STRONG:= MesBlock_Temp_1[ 7], Word_WEAK:= MesBlock_Temp_1[8], SIGNED:=TRUE, FIX:=0 , SIZE:=2, VAR_OUT:=MesDataExd.MesIdc_Group3);
		MW(WORD_STRONG:= MesBlock_Temp_1[ 9], Word_WEAK:= MesBlock_Temp_1[10], SIGNED:=TRUE, FIX:=0 , SIZE:=2, VAR_OUT:=MesDataExd.MesData.MesIdc);
		MW(WORD_STRONG:= MesBlock_Temp_1[ 11], Word_WEAK:= MesBlock_Temp_1[12], SIGNED:=TRUE, FIX:=0 , SIZE:=2, VAR_OUT:=MesDataExd.MesData.MesPdc);
		MW(WORD_STRONG:= MesBlock_Temp_1[ 13], Word_WEAK:= MesBlock_Temp_1[14], SIGNED:=TRUE, FIX:=1 , SIZE:=2, VAR_OUT:=MesDataExd.MesUdc_Group1);
		MW(WORD_STRONG:= MesBlock_Temp_1[ 15], Word_WEAK:= MesBlock_Temp_1[16], SIGNED:=TRUE, FIX:=1 , SIZE:=2, VAR_OUT:=MesDataExd.MesUdc_Group2);
		MW(WORD_STRONG:= MesBlock_Temp_1[ 17], Word_WEAK:= MesBlock_Temp_1[18], SIGNED:=TRUE, FIX:=1 , SIZE:=2, VAR_OUT:=MesDataExd.MesUdc_Group3);
		MW(WORD_STRONG:= MesBlock_Temp_1[ 19], Word_WEAK:= MesBlock_Temp_1[20], SIGNED:=TRUE, FIX:=0 , SIZE:=2, VAR_OUT:=MesDataExd.MesI1);
		MW(WORD_STRONG:= MesBlock_Temp_1[ 21], Word_WEAK:= MesBlock_Temp_1[22], SIGNED:=TRUE, FIX:=0 , SIZE:=2, VAR_OUT:=MesDataExd.MesI2);
		MW(WORD_STRONG:= MesBlock_Temp_1[ 23], Word_WEAK:= MesBlock_Temp_1[24], SIGNED:=TRUE, FIX:=0 , SIZE:=2, VAR_OUT:=MesDataExd.MesI3);
		MW(WORD_STRONG:= MesBlock_Temp_1[ 25], Word_WEAK:= MesBlock_Temp_1[26], SIGNED:=TRUE, FIX:=4 , SIZE:=2, VAR_OUT:=MesDataExd.MesData.MesCosPhi);
		MW(WORD_STRONG:= MesBlock_Temp_1[ 27], Word_WEAK:= MesBlock_Temp_1[28], SIGNED:=TRUE, FIX:=0 , SIZE:=2, VAR_OUT:=MesDataExd.MesData.MesS);
		MW(WORD_STRONG:= MesBlock_Temp_1[ 29], Word_WEAK:= MesBlock_Temp_1[30], SIGNED:=TRUE, FIX:=0 , SIZE:=2, VAR_OUT:=MesDataExd.MesData.MesP);
		MW(WORD_STRONG:= MesBlock_Temp_1[ 31], Word_WEAK:= MesBlock_Temp_1[32], SIGNED:=TRUE, FIX:=0 , SIZE:=2, VAR_OUT:=MesDataExd.MesData.MesQ);
		MW(WORD_STRONG:= MesBlock_Temp_1[ 33], Word_WEAK:= MesBlock_Temp_1[34], SIGNED:=TRUE, FIX:=1 , SIZE:=2, VAR_OUT:=MesDataExd.MesU12);
		MW(WORD_STRONG:= MesBlock_Temp_1[ 35], Word_WEAK:= MesBlock_Temp_1[36], SIGNED:=TRUE, FIX:=1 , SIZE:=2, VAR_OUT:=MesDataExd.MesU23);
		MW(WORD_STRONG:= MesBlock_Temp_1[ 37], Word_WEAK:= MesBlock_Temp_1[38], SIGNED:=TRUE, FIX:=1 , SIZE:=2, VAR_OUT:=MesDataExd.MesU31);
		MW(WORD_STRONG:= MesBlock_Temp_1[ 39], Word_WEAK:= MesBlock_Temp_1[40], SIGNED:=TRUE, FIX:=2 , SIZE:=2, VAR_OUT:=MesDataExd.MesData.MesFreq);
		MW(WORD_STRONG:= MesBlock_Temp_1[ 41], Word_WEAK:= MesBlock_Temp_1[42], SIGNED:=TRUE, FIX:=1 , SIZE:=2, VAR_OUT:=MesDataExd.MesTemp_CabAC);
		MW(WORD_STRONG:= MesBlock_Temp_1[ 43], Word_WEAK:= MesBlock_Temp_1[44], SIGNED:=TRUE, FIX:=1 , SIZE:=2, VAR_OUT:=MesDataExd.MesTemp_CabDC);
		MW(WORD_STRONG:= MesBlock_Temp_1[ 45], Word_WEAK:= MesBlock_Temp_1[46], SIGNED:=TRUE, FIX:=1 , SIZE:=2, VAR_OUT:=MesDataExd.MesTemp_CabRio);
		MW(WORD_STRONG:= MesBlock_Temp_1[ 47], Word_WEAK:= MesBlock_Temp_1[48], SIGNED:=TRUE, FIX:=1 , SIZE:=2, VAR_OUT:=MesDataExd.MesData.MesTemp);
		MW(WORD_STRONG:= MesBlock_Temp_1[ 49], Word_WEAK:= MesBlock_Temp_1[50], SIGNED:=TRUE, FIX:=1 , SIZE:=2, VAR_OUT:=MesDataExd.MesTemp_Igbt);
		MW(WORD_STRONG:= MesBlock_Temp_1[ 51], Word_WEAK:= MesBlock_Temp_1[52], SIGNED:=TRUE, FIX:=1 , SIZE:=2, VAR_OUT:=MesDataExd.MesTemp_Pcb);
		MW(WORD_STRONG:= MesBlock_Temp_1[ 53], Word_WEAK:= MesBlock_Temp_1[54], SIGNED:=TRUE, FIX:=1 , SIZE:=2, VAR_OUT:=MesDataExd.MesTemp_Ext);
		MW(WORD_STRONG:= MesBlock_Temp_1[ 55], Word_WEAK:= MesBlock_Temp_1[56], SIGNED:=TRUE, FIX:=1 , SIZE:=2, VAR_OUT:=MesDataExd.MesTemp_Transfo);
		MW_U(Word_WEAK:= MesBlock_Temp_1[ 57], WORD_STRONG:= MesBlock_Temp_1[58], VAR_OUT:=MesDataExd.MesID_DC1State);
		MW_U(Word_WEAK:= MesBlock_Temp_1[ 59], WORD_STRONG:= MesBlock_Temp_1[60], VAR_OUT:=MesDataExd.MesID_DC2State);
		MW_U(Word_WEAK:= MesBlock_Temp_1[ 61], WORD_STRONG:= MesBlock_Temp_1[62], VAR_OUT:=MesDataExd.MesID_DC3State);
		MW_U(Word_WEAK:= MesBlock_Temp_1[ 63], WORD_STRONG:= MesBlock_Temp_1[64], VAR_OUT:=MesDataExd.MesID_ACState);
		MW_U(Word_WEAK:= MesBlock_Temp_1[ 67], WORD_STRONG:= MesBlock_Temp_1[68], VAR_OUT:=MesDataExd.MesID_CapaState);
		MW_U(Word_WEAK:= MesBlock_Temp_1[ 69], WORD_STRONG:= MesBlock_Temp_1[70], VAR_OUT:=MesDataExd.MesID_PreChargeState);
		MW(WORD_STRONG:= MesBlock_Temp_1[ 71], Word_WEAK:= MesBlock_Temp_1[72], SIGNED:=FALSE, FIX:=0 , SIZE:=2, VAR_OUT:=MesDataExd.MesFeedTm);
		MW(WORD_STRONG:= MesBlock_Temp_1[ 73], Word_WEAK:= MesBlock_Temp_1[74], SIGNED:=FALSE, FIX:=0 , SIZE:=2, VAR_OUT:=MesDataExd.MesWorkingHr);
		MW(WORD_STRONG:= MesBlock_Temp_1[ 75], Word_WEAK:= MesBlock_Temp_1[76], SIGNED:=TRUE, FIX:=2 , SIZE:=2, VAR_OUT:=MesDataExd.MesEdcDischarge_Tot);
		MW(WORD_STRONG:= MesBlock_Temp_1[ 77], Word_WEAK:= MesBlock_Temp_1[78], SIGNED:=TRUE, FIX:=2 , SIZE:=2, VAR_OUT:=MesDataExd.MesEActProd_Tot);
		MW(WORD_STRONG:= MesBlock_Temp_1[ 79], Word_WEAK:= MesBlock_Temp_1[80], SIGNED:=TRUE, FIX:=2 , SIZE:=2, VAR_OUT:=MesDataExd.MesEdcDischarge_Day);
		MW(WORD_STRONG:= MesBlock_Temp_1[ 81], Word_WEAK:= MesBlock_Temp_1[82], SIGNED:=TRUE, FIX:=2 , SIZE:=2, VAR_OUT:=MesDataExd.MesEActProd_Day);
		MW(WORD_STRONG:= MesBlock_Temp_1[ 83], Word_WEAK:= MesBlock_Temp_1[84], SIGNED:=FALSE, FIX:=0 , SIZE:=2, VAR_OUT:=MesDataExd.MesWorkingHr_Fan1);
		MW(WORD_STRONG:= MesBlock_Temp_1[ 85], Word_WEAK:= MesBlock_Temp_1[86], SIGNED:=FALSE, FIX:=0 , SIZE:=2, VAR_OUT:=MesDataExd.MesWorkingHr_Fan2);
		MW(WORD_STRONG:= MesBlock_Temp_1[ 87], Word_WEAK:= MesBlock_Temp_1[88], SIGNED:=FALSE, FIX:=0 , SIZE:=2, VAR_OUT:=MesDataExd.MesWorkingHr_BridgeFan);
		MW(WORD_STRONG:= MesBlock_Temp_1[ 89], Word_WEAK:= MesBlock_Temp_1[90], SIGNED:=FALSE, FIX:=0 , SIZE:=2, VAR_OUT:=MesDataExd.MesWorkingHr_Heater);
		MW(WORD_STRONG:= MesBlock_Temp_1[ 91], Word_WEAK:= MesBlock_Temp_1[92], SIGNED:=FALSE, FIX:=0 , SIZE:=2, VAR_OUT:=MesDataExd.MesWorkingHr_Heater2);
		MW_U(Word_WEAK:= MesBlock_Temp_1[ 93], WORD_STRONG:= MesBlock_Temp_1[94], VAR_OUT:=MesDataExd.MesID_ErrorLocation);
		MW_U(Word_WEAK:= MesBlock_Temp_1[ 95], WORD_STRONG:= MesBlock_Temp_1[96], VAR_OUT:=MesDataExd.MesID_ErrorState);
		
		MW(WORD_STRONG:= MesBlock_Temp_1[ 97], Word_WEAK:= MesBlock_Temp_1[98], SIGNED:=FALSE, FIX:=0 , SIZE:=2, VAR_OUT:=MesDataExd.MesEventID);
		
		MW_U(Word_WEAK:= MesBlock_Temp_1[ 99], WORD_STRONG:= MesBlock_Temp_1[100], VAR_OUT:=MesDataExd.MesData.MesState_Inv);
		MW_U(Word_WEAK:= MesBlock_Temp_1[ 101], WORD_STRONG:= MesBlock_Temp_1[102], VAR_OUT:=MesDataExd.MesID_StartKeyState);
		
		MW(WORD_STRONG:= MesBlock_Temp_1[ 103], Word_WEAK:= MesBlock_Temp_1[104], SIGNED:=TRUE, FIX:=1 , SIZE:=2, VAR_OUT:=MesDataExd.MesTime_GridConnWait);
		
		MW_U(Word_WEAK:= MesBlock_Temp_1[ 107], WORD_STRONG:= MesBlock_Temp_1[108], VAR_OUT:=MesDataExd.MesID_GFDIState);
		MW(WORD_STRONG:= MesBlock_Temp_1[ 109], Word_WEAK:= MesBlock_Temp_1[110], SIGNED:=TRUE, FIX:=0 , SIZE:=2, VAR_OUT:=MesDataExd.MesSetptP);
		MW(WORD_STRONG:= MesBlock_Temp_1[ 111], Word_WEAK:= MesBlock_Temp_1[112], SIGNED:=TRUE, FIX:=1 , SIZE:=2, VAR_OUT:=MesDataExd.MesSetptSmax);
		MW(WORD_STRONG:= MesBlock_Temp_1[ 113], Word_WEAK:= MesBlock_Temp_1[114], SIGNED:=TRUE, FIX:=0 , SIZE:=2, VAR_OUT:=MesDataExd.MesSetptQ);
		MW(WORD_STRONG:= MesBlock_Temp_1[ 115], Word_WEAK:= MesBlock_Temp_1[116], SIGNED:=TRUE, FIX:=4 , SIZE:=2, VAR_OUT:=MesDataExd.MesSetptCosPhi);
		MW_U(Word_WEAK:= MesBlock_Temp_1[ 117], WORD_STRONG:= MesBlock_Temp_1[118], VAR_OUT:=MesDataExd.MesID_AlarmGas_Transfo);
		MW_U(Word_WEAK:= MesBlock_Temp_1[ 119], WORD_STRONG:= MesBlock_Temp_1[120], VAR_OUT:=MesDataExd.MesID_AlarmTemp_Transfo);
		MW_U(Word_WEAK:= MesBlock_Temp_1[ 121], WORD_STRONG:= MesBlock_Temp_1[122], VAR_OUT:=MesDataExd.MesID_AlarmOilLevel_Transfo);
		MW_U(Word_WEAK:= MesBlock_Temp_1[ 123], WORD_STRONG:= MesBlock_Temp_1[124], VAR_OUT:=MesDataExd.MesIDWarningTemp_Transfo);
		
		
		
		
	// Block 2 
		MW(WORD_STRONG:= MesBlock_Temp_2[ 1], Word_WEAK:= MesBlock_Temp_2[2], SIGNED:=TRUE, FIX:=1 , SIZE:=2, VAR_OUT:=MesDataExd.MesTemp_Igbt1);
		MW(WORD_STRONG:= MesBlock_Temp_2[ 7], Word_WEAK:= MesBlock_Temp_2[8], SIGNED:=TRUE, FIX:=1 , SIZE:=2, VAR_OUT:=MesDataExd.MesTemp_Pcb1);
		MW(WORD_STRONG:= MesBlock_Temp_2[ 9], Word_WEAK:= MesBlock_Temp_2[10], SIGNED:=TRUE, FIX:=1 , SIZE:=2, VAR_OUT:=MesDataExd.MesTemp_Pcb2);
		MW(WORD_STRONG:= MesBlock_Temp_2[ 11], Word_WEAK:= MesBlock_Temp_2[12], SIGNED:=TRUE, FIX:=1 , SIZE:=2, VAR_OUT:=MesDataExd.MesTemp_Pcb3);
		MW(WORD_STRONG:= MesBlock_Temp_2[ 13], Word_WEAK:= MesBlock_Temp_2[14], SIGNED:=TRUE, FIX:=2 , SIZE:=2, VAR_OUT:=MesDataExd.MesEAct_PreviousDay);
		MW(WORD_STRONG:= MesBlock_Temp_2[ 15], Word_WEAK:= MesBlock_Temp_2[16], SIGNED:=FALSE, FIX:=0 , SIZE:=2, VAR_OUT:=MesDataExd.MesWorkingHr_Cpu);
		MW(WORD_STRONG:= MesBlock_Temp_2[ 17], Word_WEAK:= MesBlock_Temp_2[18], SIGNED:=TRUE, FIX:=1 , SIZE:=2, VAR_OUT:=MesDataExd.MesData.MesInsuResistor);
		MW(WORD_STRONG:= MesBlock_Temp_2[ 19], Word_WEAK:= MesBlock_Temp_2[20], SIGNED:=TRUE, FIX:=2 , SIZE:=2, VAR_OUT:=MesDataExd.MesPressure_Transfo);
		
		MW_U(Word_WEAK:= MesBlock_Temp_2[ 21], WORD_STRONG:= MesBlock_Temp_2[22], VAR_OUT:=MesDataExd.MesID_PresMonitorState_Transfo);
		
		MW(WORD_STRONG:= MesBlock_Temp_2[ 23], 									SIGNED:=FALSE, FIX:=0 , SIZE:=1, VAR_OUT:=MesDataExd.MesState_BackFeedMode);
		MW(WORD_STRONG:= MesBlock_Temp_2[ 24], Word_WEAK:= MesBlock_Temp_2[25], SIGNED:=TRUE, FIX:=1 , SIZE:=2, VAR_OUT:=MesDataExd.MesIdc_BackFeed);
		
		MW(WORD_STRONG:= MesBlock_Temp_2[ 28], Word_WEAK:= MesBlock_Temp_2[29], SIGNED:=TRUE, FIX:=2 , SIZE:=2, VAR_OUT:=MesDataExd.MesEdcCharge_Tot);
		MW(WORD_STRONG:= MesBlock_Temp_2[ 30], Word_WEAK:= MesBlock_Temp_2[31], SIGNED:=TRUE, FIX:=2 , SIZE:=2, VAR_OUT:=MesDataExd.MesEActCons_Tot);
		MW(WORD_STRONG:= MesBlock_Temp_2[ 32], Word_WEAK:= MesBlock_Temp_2[33], SIGNED:=TRUE, FIX:=2 , SIZE:=2, VAR_OUT:=MesDataExd.MesEdcCharge_Day);
		MW(WORD_STRONG:= MesBlock_Temp_2[ 34], Word_WEAK:= MesBlock_Temp_2[35], SIGNED:=TRUE, FIX:=2 , SIZE:=2, VAR_OUT:=MesDataExd.MesEActCons_Day);
		MW(WORD_STRONG:= MesBlock_Temp_2[ 36], Word_WEAK:= MesBlock_Temp_2[37], SIGNED:=TRUE, FIX:=1 , SIZE:=2, VAR_OUT:=MesDataExd.MesSetptUdc);
		MW(WORD_STRONG:= MesBlock_Temp_2[ 40], Word_WEAK:= MesBlock_Temp_2[41], SIGNED:=TRUE, FIX:=4 , SIZE:=2, VAR_OUT:=MesDataExd.MesSetptU);
		
		MW(WORD_STRONG:= MesBlock_Temp_2[ 47], Word_WEAK:= MesBlock_Temp_2[48], SIGNED:=TRUE, FIX:=2 , SIZE:=2, VAR_OUT:=MesDataExd.MesSetptFreq);
		MW(WORD_STRONG:= MesBlock_Temp_2[ 49], Word_WEAK:= MesBlock_Temp_2[50], SIGNED:=TRUE, FIX:=4 , SIZE:=2, VAR_OUT:=MesDataExd.MesPconnected);
		MW(WORD_STRONG:= MesBlock_Temp_2[ 51], Word_WEAK:= MesBlock_Temp_2[52], SIGNED:=TRUE, FIX:=4 , SIZE:=2, VAR_OUT:=MesDataExd.MesQconnected);
		
		MW_U(Word_WEAK:= MesBlock_Temp_2[ 53], WORD_STRONG:= MesBlock_Temp_2[54], VAR_OUT:=MesDataExd.MesID_Derating);
		MW_U(Word_WEAK:= MesBlock_Temp_2[ 55], WORD_STRONG:= MesBlock_Temp_2[56], VAR_OUT:=MesDataExd.MesID_Off);
		
		MW(WORD_STRONG:= MesBlock_Temp_2[ 57], Word_WEAK:= MesBlock_Temp_2[58], SIGNED:=FALSE, FIX:=0 , SIZE:=2, VAR_OUT:=MesDataExd.MesTime_SelfTestWait);
		MW(WORD_STRONG:= MesBlock_Temp_2[ 59], SIGNED:=FALSE, FIX:=0 , SIZE:=1, VAR_OUT:=MesDataExd.MesID_WarningFloatCtrl);
		MW(WORD_STRONG:= MesBlock_Temp_2[ 60], SIGNED:=FALSE, FIX:=0 , SIZE:=1, VAR_OUT:=MesDataExd.MesID_ErrorFloatCtrl);
		MW(WORD_STRONG:= MesBlock_Temp_2[ 61], Word_WEAK:= MesBlock_Temp_2[62], SIGNED:=TRUE, FIX:=0 , SIZE:=2, VAR_OUT:=MesDataExd.MesData.ParamPn);
		MW(WORD_STRONG:= MesBlock_Temp_2[ 63], SIGNED:=TRUE, FIX:=2 , SIZE:=1, VAR_OUT:=MesDataExd.MesIGnd);
		MW(WORD_STRONG:= MesBlock_Temp_2[ 64], SIGNED:=TRUE, FIX:=2 , SIZE:=1, VAR_OUT:=MesDataExd.MesIGnd_LastError);
		
		MW(WORD_STRONG:= MesBlock_Temp_2[ 65], Word_WEAK:= MesBlock_Temp_2[66], SIGNED:=FALSE, FIX:=0 , SIZE:=2, VAR_OUT:=MesDataExd.MesEventID1);
		MW_U(Word_WEAK:= MesBlock_Temp_2[ 67], WORD_STRONG:= MesBlock_Temp_2[68], VAR_OUT:=MesDataExd.MesID_ErrorLocation1);
		MW(WORD_STRONG:= MesBlock_Temp_2[ 69], Word_WEAK:= MesBlock_Temp_2[70], SIGNED:=FALSE, FIX:=0 , SIZE:=2, VAR_OUT:=MesDataExd.MesEventID2);
		MW_U(Word_WEAK:= MesBlock_Temp_2[ 71], WORD_STRONG:= MesBlock_Temp_2[72], VAR_OUT:=MesDataExd.MesID_ErrorLocation2);
		MW(WORD_STRONG:= MesBlock_Temp_2[ 73], Word_WEAK:= MesBlock_Temp_2[74], SIGNED:=FALSE, FIX:=0 , SIZE:=2, VAR_OUT:=MesDataExd.MesEventID3);
		MW_U(Word_WEAK:= MesBlock_Temp_2[ 75], WORD_STRONG:= MesBlock_Temp_2[76], VAR_OUT:=MesDataExd.MesID_ErrorLocation3);
		MW(WORD_STRONG:= MesBlock_Temp_2[ 77], Word_WEAK:= MesBlock_Temp_2[78], SIGNED:=FALSE, FIX:=0 , SIZE:=2, VAR_OUT:=MesDataExd.MesEventID4);
		MW_U(Word_WEAK:= MesBlock_Temp_2[ 79], WORD_STRONG:= MesBlock_Temp_2[80], VAR_OUT:=MesDataExd.MesID_ErrorLocation4);
		MW(WORD_STRONG:= MesBlock_Temp_2[ 81], Word_WEAK:= MesBlock_Temp_2[82], SIGNED:=FALSE, FIX:=0 , SIZE:=2, VAR_OUT:=MesDataExd.MesEventID5);
		MW_U(Word_WEAK:= MesBlock_Temp_2[ 83], WORD_STRONG:= MesBlock_Temp_2[84], VAR_OUT:=MesDataExd.MesID_ErrorLocation5);
		MW(WORD_STRONG:= MesBlock_Temp_2[ 85], Word_WEAK:= MesBlock_Temp_2[86], SIGNED:=FALSE, FIX:=0 , SIZE:=2, VAR_OUT:=MesDataExd.MesEventID6);
		MW_U(Word_WEAK:= MesBlock_Temp_2[ 87], WORD_STRONG:= MesBlock_Temp_2[88], VAR_OUT:=MesDataExd.MesID_ErrorLocation6);
		MW(WORD_STRONG:= MesBlock_Temp_2[ 89], Word_WEAK:= MesBlock_Temp_2[90], SIGNED:=FALSE, FIX:=0 , SIZE:=2, VAR_OUT:=MesDataExd.MesEventID7);
		MW_U(Word_WEAK:= MesBlock_Temp_2[ 91], WORD_STRONG:= MesBlock_Temp_2[92], VAR_OUT:=MesDataExd.MesID_ErrorLocation7);
		MW(WORD_STRONG:= MesBlock_Temp_2[ 93], Word_WEAK:= MesBlock_Temp_2[94], SIGNED:=FALSE, FIX:=0 , SIZE:=2, VAR_OUT:=MesDataExd.MesEventID8);
		MW_U(Word_WEAK:= MesBlock_Temp_2[ 95], WORD_STRONG:= MesBlock_Temp_2[96], VAR_OUT:=MesDataExd.MesID_ErrorLocation8);
		MW(WORD_STRONG:= MesBlock_Temp_2[ 97], Word_WEAK:= MesBlock_Temp_2[98], SIGNED:=FALSE, FIX:=0 , SIZE:=2, VAR_OUT:=MesDataExd.MesEventID9);
		MW_U(Word_WEAK:= MesBlock_Temp_2[ 99], WORD_STRONG:= MesBlock_Temp_2[100], VAR_OUT:=MesDataExd.MesID_ErrorLocation9);
		MesDataExd.MesEventID10:=MesBlock_Temp_2[101];
		MesDataExd.MesID_ErrorLocation10:=MesBlock_Temp_2[103];
		
		(*
	// Block 3  ( Inputs  )MesIdc_input1
		MW(WORD_STRONG:= MesBlock_Temp_3[ 1], SIGNED:=TRUE, FIX:=1 , SIZE:=1, VAR_OUT:=MesDataExd.MesIdc_input1);
		MW(WORD_STRONG:= MesBlock_Temp_3[ 2], SIGNED:=TRUE, FIX:=1 , SIZE:=1, VAR_OUT:=MesDataExd.MesIdc_input2);
		MW(WORD_STRONG:= MesBlock_Temp_3[ 3], SIGNED:=TRUE, FIX:=1 , SIZE:=1, VAR_OUT:=MesDataExd.MesIdc_input3);
		MW(WORD_STRONG:= MesBlock_Temp_3[ 4], SIGNED:=TRUE, FIX:=1 , SIZE:=1, VAR_OUT:=MesDataExd.MesIdc_input4);
		MW(WORD_STRONG:= MesBlock_Temp_3[ 5], SIGNED:=TRUE, FIX:=1 , SIZE:=1, VAR_OUT:=MesDataExd.MesIdc_input5);
		MW(WORD_STRONG:= MesBlock_Temp_3[ 6], SIGNED:=TRUE, FIX:=1 , SIZE:=1, VAR_OUT:=MesDataExd.MesIdc_input6);
		MW(WORD_STRONG:= MesBlock_Temp_3[ 7], SIGNED:=TRUE, FIX:=1 , SIZE:=1, VAR_OUT:=MesDataExd.MesIdc_input7);
		//MW(WORD_STRONG:= MesBlock_Temp_3[ 8], SIGNED:=TRUE, FIX:=1 , SIZE:=1, VAR_OUT:=MesDataExd.MesIdc_input8); free
		MW(WORD_STRONG:= MesBlock_Temp_3[ 9], SIGNED:=TRUE, FIX:=1 , SIZE:=1, VAR_OUT:=MesDataExd.MesIdc_input9);
		MW(WORD_STRONG:= MesBlock_Temp_3[ 10], SIGNED:=TRUE, FIX:=1 , SIZE:=1, VAR_OUT:=MesDataExd.MesIdc_input10);
		MW(WORD_STRONG:= MesBlock_Temp_3[ 11], SIGNED:=TRUE, FIX:=1 , SIZE:=1, VAR_OUT:=MesDataExd.MesIdc_input11);
		MW(WORD_STRONG:= MesBlock_Temp_3[ 12], SIGNED:=TRUE, FIX:=1 , SIZE:=1, VAR_OUT:=MesDataExd.MesIdc_input12);
		
		
	// Block 4 ( Inputs ) 
		MW(WORD_STRONG:= MesBlock_Temp_4[ 1], SIGNED:=TRUE, FIX:=1 , SIZE:=1, VAR_OUT:=MesDataExd.MesIdc_input13);
		MW(WORD_STRONG:= MesBlock_Temp_4[ 2], SIGNED:=TRUE, FIX:=1 , SIZE:=1, VAR_OUT:=MesDataExd.MesIdc_input14);
		MW(WORD_STRONG:= MesBlock_Temp_4[ 3], SIGNED:=TRUE, FIX:=1 , SIZE:=1, VAR_OUT:=MesDataExd.MesIdc_input15);
		//MW(WORD_STRONG:= MesBlock_Temp_4[ 4], SIGNED:=TRUE, FIX:=1 , SIZE:=1, VAR_OUT:=MesDataExd.MesIdc_input16);
		MW(WORD_STRONG:= MesBlock_Temp_4[ 5], SIGNED:=TRUE, FIX:=1 , SIZE:=1, VAR_OUT:=MesDataExd.MesIdc_input17);
		MW(WORD_STRONG:= MesBlock_Temp_4[ 6], SIGNED:=TRUE, FIX:=1 , SIZE:=1, VAR_OUT:=MesDataExd.MesIdc_input18);
		MW(WORD_STRONG:= MesBlock_Temp_4[ 7], SIGNED:=TRUE, FIX:=1 , SIZE:=1, VAR_OUT:=MesDataExd.MesIdc_input19);
		MW(WORD_STRONG:= MesBlock_Temp_4[ 8], SIGNED:=TRUE, FIX:=1 , SIZE:=1, VAR_OUT:=MesDataExd.MesIdc_input20);
		MW(WORD_STRONG:= MesBlock_Temp_4[ 9], SIGNED:=TRUE, FIX:=1 , SIZE:=1, VAR_OUT:=MesDataExd.MesIdc_input21);
		MW(WORD_STRONG:= MesBlock_Temp_4[ 10], SIGNED:=TRUE, FIX:=1 , SIZE:=1, VAR_OUT:=MesDataExd.MesIdc_input22);
		MW(WORD_STRONG:= MesBlock_Temp_4[ 11], SIGNED:=TRUE, FIX:=1 , SIZE:=1, VAR_OUT:=MesDataExd.MesIdc_input23);
		//MW(WORD_STRONG:= MesBlock_Temp_4[ 12], SIGNED:=TRUE, FIX:=1 , SIZE:=1, VAR_OUT:=MesDataExd.MesIdc_input24);
		*)
		
		
	// Data calculation 
		MesDataExd.MesData.MesCurtl  		:=   MesDataExd.MesID_Derating > 21584 ; 
		MesDataExd.MesDAta.MesOpened_Ac 	:= MesDataExd.MesID_ACState = 311 ; 
		MesDataExd.MesDAta.MesOpened_Dc 	:=  MesDataExd.MesID_DC1State = 311 AND MesDataExd.MesID_DC2State = 311 AND MesDataExd.MesID_DC3State = 311 ; 
		MesDataExd.Mesdata.MesU				:= (MesDataExd.MesU12 + MesDataExd.MesU23 + MesDataExd.MesU31) / 3 ; 
		MesDataExd.MesData.ParamPn	:= ParamPn ; 


END_IF
END_METHOD

METHOD M_StartStop 
VAR_INPUT
END_VAR
VAR
	KK : UINT;
	AX_ADR_MB			: WORD := 0;
	AX_QTY_MB			: ARRAY[1..2] OF BYTE := [2, 2];
	MotStart			: WORD := 309; // operation 
	MotStop				: WORD := 381; // stop
	
END_VAR
SUPER^.M_StartStop() ; 
FB_ModbusWrite[1](WriteCmd := FALSE);

//Read the setpoints
	// Evaluate the cmd given 
Trig_Local_Start(CLK:=IN_CmdStart_Local);
Trig_Local_Stop(CLK:=IN_CmdStop_Local);
Trig_Start(CLK:=IN_CmdStart AND RS_StartStop_Local.Q1 );
Trig_Stop(CLK:=IN_CmdStop);

RS_StartStop_Local(SET:=Trig_Local_Start.Q,Reset1:= Trig_Local_Stop.Q); // TRUE START, FALSE STOP
RS_StartStop(SET:=Trig_Start.Q,Reset1 := Trig_Stop.Q OR NOT RS_StartStop_Local.Q1 ); // TRUE START, FALSE STOP


//CalCP_CMD_StartStop := RS_StartStop.Q1 <> MesState.1 ; 

MesDataExd.MesData.OUT_CmdStart := RS_StartStop.Q1 ; 
MesDataExd.MesData.OUT_CmdStop := NOT RS_StartStop.Q1  ;


	IF RS_StartStop.Q1 THEN
		MesBlockWrite3_Temp[1] := 0;
		MesBlockWrite3_Temp[2] := MotStart;
	ELSE 
		MesBlockWrite3_Temp[1] := 0;
		MesBlockWrite3_Temp[2] := MotStop;
	END_IF

	
	FB_ModbusWrite[3]
	(
		pSrcAddr := ADR (MesBlockWrite3_Temp),
		sIPAddr := ParamIPAddress,
		tTimeout := ParamTimeout,
		nMBAddr := AX_ADR_MB,
		nTCPport := ParamTCPPort,
		cbLength := SIZEOF(MesBlockWrite3_Temp),
		nQuantity := 2,
		nUnitID := ParamUnitID,
		WriteCmd := (Trig_Start.Q OR Trig_Stop.Q OR Trig_Local_Start.Q OR Trig_Local_Stop.Q)AND MesDataExd.MesData.MesCP_Write ,
		Reset := CmdClearFault_G,
		ErrorId => AX_ModbusWriteAlarmId[1],
		ModbusWriteAlarm => AX_ModbusWriteAlarm[1]
	);
END_METHOD

METHOD M_StateManager
//////////////////
// Detect which is the state of the inverter. IF loss of communication MesState =0 , the last inverter state is kept .  
/////////////////

VAR 
	// Method local variables (reinitialized at each cycle) 

	
END_VAR
MesDataExd.MesData.MesState 			:= 0  ; 
//O=Stopped, 1 = MPPT, 2 = Sleeping, 3 = Starting, 4 = Throttled, 5 = Shutting down, 6 = Fault, 7 = Standby


// Stopped
IF 		
		MesDataExd.MesData.MesState_Inv = 381 OR  //Stop
		MesDataExd.MesData.MesState_Inv = 1394 OR  //Wait AC
		MesDataExd.MesData.MesState_Inv = 3524 OR  // Connect  AC
		MesDataExd.MesData.MesState_Inv = 1393 OR  // Wait DC
		MesDataExd.MesData.MesState_Inv = 3525  	// Connect DC
THEN // 
	MesDataExd.MesData.MesState.0 := TRUE;		
ELSIF MesDataExd.MesData.MesState_Inv = 3526 AND (MesDataExd.MesID_Derating = 21594 OR  MesDataExd.MesID_Derating = 973) THEN //GridFeed and maxW
	MesDataExd.MesData.MesState.1 := TRUE;
ELSIF 	MesDataExd.MesData.MesState_Inv = 1787 OR //Init
	MesDataExd.MesData.MesState_Inv = 375  //Selftest
 THEN
	MesDataExd.MesData.MesState.3 := TRUE;
ELSIF MesDataExd.MesData.MesState_Inv = 3526 AND (MesDataExd.MesID_Derating <> 21594 OR  MesDataExd.MesID_Derating <> 973) THEN //GridFeed and not maxW
	MesDataExd.MesData.MesState.4 := TRUE;
ELSIF 
		MesDataExd.MesData.MesState_Inv = 3530   OR	//RampDown
		MesDataExd.MesData.MesState_Inv = 1469	// ShutDown
THEN
	MesDataExd.MesData.MesState.5 := TRUE;

ELSIF 
		MesDataExd.MesData.MesState_Inv = 1392   // Error
THEN
	MesDataExd.MesData.MesState.6 := TRUE;

ELSIF 		MesDataExd.MesData.MesState_Inv = 3528  
THEN
	MesDataExd.MesData.MesState.7 := TRUE;

END_IF

SUPER^.M_StateManager() ;
END_METHOD

END_FUNCTION_BLOCK

// ---- 00_FunctionsBlocks/Beckhoff/Communication/ModbusTCP/FB_ModbusReadInputRegs.TcPOU
FUNCTION_BLOCK FB_ModbusReadInputRegs
////////////////// 
// Read Modbus TCP/IP on Rising Edge of Trigger ClockRead. Returns alarm and stop modbus Read after three consecutive Modbus attempts that failed. 
//////////////////

VAR_INPUT
	
	// Modbus ReadRegs FB inputs
	pDestAddr 	: POINTER TO BYTE ; // Pointer to variable in which the read data have to be stored
	sIPAddr 	: STRING(15);		// Modbus server device IP adress
	tTimeout 	: TIME;				// Timeout
	
	nTCPport	: UINT:= 502;		// TCP Port
	
	nQuantity 	: WORD;				// Quantity of words to be read
	nMBAddr 	: WORD ;			// Starting Register adress
	
	cbLength 	: UDINT;			// Length of variable to host the read data
	nUnitID 	: BYTE;				// Unit ID in case of serial connexion after modbus server. Usually equals to 1
	
	ClockRead	: BOOL; 			// Rising Edge Modbus Trigger
	Reset		: BOOL; 			// Reset Trigger to clean alarm and counter.
	
	ParamTimeRetry 			: TIME:=T#30S;				//Time to wait before a retry
	ParamNbAlms				: INT := 3;				// Parameter for the number of retries before the alarme
	ParamEnableRetryPause	: BOOL ; 
	
END_VAR

VAR_OUTPUT
	ErrorId			: UDINT;	// Error Id returned by FB ( see ADS error Code ) . 
	OUT_Completed	: BOOL ; // Reading completed successfully . 
	Busy			: BOOL ;	// FB busy to proceed command
	ModbusReadAlarm	: BOOL; 	// Alarm if three modbus attempt failed.
	
END_VAR

VAR
	R_TRIG 				: R_TRIG; 			// Rising edge detection for the trigger.
	FB_MBReadInputRegs 	: FB_MBReadInputRegs; 	// Multiple registers reading
	
	Step				: INT; 				// Grafcet step
	AlarmCounter		: INT; 				// Alarm Counter. Incremennted if modbus errOR  Alarm if counter =3 , resetable.  
	TempoRetry      		: TP;

	bRetry          		: BOOL:= FALSE; 			// Boolean to denote the retries	
	
END_VAR

// ALARM MANAGEMENT //
TempoRetry(PT := ParamTimeRetry);
	IF AlarmCounter=3 THEN 
		ModbusReadAlarm 	:=TRUE;
		bRetry := SEL(ParamEnableRetryPause , FALSE ,  TRUE);		// False = disable retry 		
	ELSE
		ModbusReadAlarm := FALSE;
		ErrorId			:= 0;
		bRetry := FALSE;		// False = disable retry 
	END_IF

OUT_Completed := FALSE ; 

// MODBUS SEQUENCE //
CASE Step OF 
	0:
		R_TRIG(CLK :=ClockRead);
		IF R_TRIG.Q THEN 
			Step :=1;
			Busy := TRUE;
		END_IF
	1:
	   FB_MBReadInputRegs(
	  			sIPAddr:= sIPAddr , 
				nTCPPort:= nTCPport ,
				nUnitID:= nUnitID,
				nQuantity:= nQuantity,
				nMBAddr:= nMBAddr, 
				cbLength:= cbLength, 
				pDestAddr:= pDestAddr, 
				bExecute:= TRUE,
				tTimeout:= tTimeout
				);
				
		IF NOT FB_MBReadInputRegs.bBusy AND NOT FB_MBReadInputRegs.bError THEN
			OUT_Completed := TRUE ;
			FB_MBReadInputRegs(bExecute:= FALSE);
			AlarmCounter	:=0; // Reset counter after successful modbus read. 
			Step 			:=0;
			Busy := FALSE;
		ELSIF NOT FB_MBReadInputRegs.bBusy AND FB_MBReadInputRegs.bError AND NOT(bRetry) THEN
			FB_MBReadInputRegs(bExecute:= FALSE);
			AlarmCounter 	:= MIN(AlarmCounter+1,3) ; 
			ErrorId			 :=FB_MBReadInputRegs.nErrId;
			Step 			:=0;
			Busy := FALSE;
		ELSIF NOT FB_MBReadInputRegs.bBusy AND FB_MBReadInputRegs.bError AND bRetry THEN
			step := 2;
			Busy := FALSE;		
			
		END_IF
	2: 
		TempoRetry(In:= TRUE);		// LEAVE SOME TIME BEFORE NEW ATTEMPT . 
		IF NOT(TempoRetry.Q) THEN
			TempoRetry(In:= FALSE);
			//AlarmCounter := 0;
			step := 0;
			
		END_IF	
END_CASE

// RESET //
	IF Reset THEN 
		AlarmCounter 		:= 0 ; 
		ErrorId 			:= 0 ; 
		ModbusReadAlarm 	:=FALSE;
		Reset 				:= FALSE;
	END_IF

// BUSY //
	//Busy 						:= FB_MBReadInputRegs.bBusy ;

ACTION Init:

END_ACTION

END_FUNCTION_BLOCK

// ---- 00_FunctionsBlocks/Common/DataProcessing/MergeWord/FB_MergeWordsToUint.TcPOU
FUNCTION_BLOCK FB_MergeWordsToUint
////////////////// 
// Merge two words or one word into a DINT or UDINT with big endian coding. And finally Output a Real. 
//////////////////	

VAR_IN_OUT
	VAR_OUT 		: UINT ; 	
	
END_VAR

VAR_INPUT
	WORD_STRONG 		: WORD; 			// Strong Word. Word to consider if size equals 1.
	WORD_WEAK	 		: WORD 	:= 0; 		// Weak Word. 
	

END_VAR

VAR
	VAR_AUX 		: ULINT ;			
	
END_VAR


MEMCPY(destAddr := ADR(VAR_OUT)+1*SIZEOF(WORD_STRONG), 		srcAddr := ADR(WORD_WEAK), 		n := SIZEOF(WORD_WEAK));
MEMCPY(destAddr := ADR(VAR_OUT)+0*SIZEOF(WORD_STRONG), 		srcAddr := ADR(WORD_STRONG), 	n := SIZEOF(WORD_WEAK));

END_FUNCTION_BLOCK

// ---- 01_Equipement_Library/Inverter/FB_INV_PE_HEMK.TcPOU
FUNCTION_BLOCK FB_INV_PE_HEMK EXTENDS FB_INV_Base

VAR_INPUT PERSISTENT
		ParamTcpPort				: UINT := 502;					  (* (NA) TCP port *)
		ParamIPAddress				: STRING; 						  (* (NA) Config: IP Adress of PV Inverter *)
		ParamUnitID 				: BYTE; 						  (* (NA) PE SKID Modbus Unit ID *)
		
		ParamSmax					: REAL := 3800;					  (* (kVA) Maximum apparent power of the SKID *)
		ParamID_INV					: UINT := 1;					  (* (NA) INV number 1 or 2 in the SKID *)
		ParamNbDU					: BYTE := 10; 					  (* (NA) Total Number of disconnecting units (cables wired on the PCS) *)				
		ParamNbDU_PowerCol			: ARRAY[1..3] OF BYTE := [5,5,5]; (* (NA) Number of disconnecting uits for each Power Columns *)		
		
		ParamPref_NoCom				: REAL := 100;					  (* (%) P reference defaut value in case Reset refs time different from OFF and loss of communication with PPC *)
		ParamQref_NoCom				: REAL := 0;					  (* (%) Q reference defaut value in case Reset refs time different from OFF and loss of communication with PPC *)
END_VAR

VAR_INPUT 
		IN_CmdEmergencyStop_Local	: BOOL;	
		MesDataExd		AT %Q*		: INV_PE_HEMK; 					   // (NA) Inverter Object 
END_VAR
VAR	
	// M_READ VARIABLES//		
		Trig_Local_EmergencyStop	: R_Trig;
		Trig_Reset					: R_Trig;
		FTrig_Watchdog				: F_Trig;
		Timer_Watchdog				: BOOL;
		Watchdog_CP_Write			: BOOL;
		TP_Watchdog					: TP;
		
		FB_ModbusRead	          	: ARRAY[1..20] OF FB_ModbusRead; // (NA) FB for Modbus Reading
		AX_ModbusReadAlarm			: ARRAY[1..20] OF BOOL;
		AX_ModbusReadAlarmId		: ARRAY[1..20] OF UDINT;

		FB_ModbusWrite				: ARRAY[1..9]  OF FB_ModbusWrite;
		AX_ModbusWriteAlarm			: ARRAY[1..9]  OF BOOL;
		AX_ModbusWriteAlarmId		: ARRAY[1..9]  OF UDINT;	
	
		MesBlock_Temp_1 			: ARRAY [1..120] OF WORD ; 		// (NA) Temporary Block with multiple modbus reading 
		MesBlock_Temp_2 			: ARRAY [1..120] OF WORD ; 		// (NA) Temporary Block with multiple modbus reading 
		MesBlock_Temp_3 			: ARRAY [1..120] OF WORD ; 		// (NA) Temporary Block with multiple modbus reading 
		MesBlock_Temp_4 			: ARRAY [1..120] OF WORD ; 		// (NA) Temporary Block with multiple modbus reading 
		MesBlock_Temp_5 			: ARRAY [1..120] OF WORD ; 		// (NA) Temporary Block with multiple modbus reading 
		MesBlock_Temp_6 			: ARRAY [1..120] OF WORD ; 		// (NA) Temporary Block with multiple modbus reading 
		MesBlock_Temp_7 			: ARRAY [1..120] OF WORD ; 		// (NA) Temporary Block with multiple modbus reading 
		MesBlock_Temp_8 			: ARRAY [1..CstNbPowerCol_INV_G] OF ARRAY [1..120] OF WORD ; 		// (NA) Temporary Block with multiple modbus reading 
		MesBlock_Temp_9 			: ARRAY [1..120] OF WORD ; 		// (NA) Temporary Block with multiple modbus reading
		
		
		MesBlockWrite1_Temp 		: WORD;							// (NA) Temporary Block with multiple modbus writing (Caution : Double Word variables)
		MesBlockWrite2_Temp			: ARRAY[1..3] OF WORD;			// (NA) Temporary Block with multiple modbus writing (Caution : Double Word variables)
		MesBlockWrite3_Temp			: WORD;							// (NA) Temporary Block with multiple modbus writing (Caution : Double Word variables)
		MesBlockWrite4_Temp			: ARRAY[1..10] OF WORD;			// (NA) Temporary Block with multiple modbus writing (Caution : Double Word variables)
		MesBlockWrite5_Temp			: ARRAY[1..2] OF WORD;
		MesBlockWrite6_Temp			: WORD;
		MesBlockWrite7_Temp			: ARRAY[1..2] OF WORD;
		MesBlockWrite8_Temp			: WORD;
		TON_BJ						: ARRAY[1..10] OF TON; 

		AX_QTY_MB					: ARRAY[1..8] OF WORD := [10, 		8,		120, 	12,		33, 	40,		2,		35];   		// Correction Imed : La premiere valeur était 2
		AX_ADR_MB					: ARRAY[1..8] OF WORD := [540,		637, 	1000, 	1372,	4300,	5000,	6500,	6505];		// Correction Imed : La premiere valeur était 539
	// M_STARTSTOP//
		StartStop_RTrig				: R_Trig;
              	
	// M_CP
		CalCP_CMD_StartStop			: BOOL; 						// Write command start;
END_VAR

METHOD M_AlarmManagement
//////////////////
// Manages IntelliGen Alarms
/////////////////

VAR 
	// Method local variables (reinitialized at each cycle) 
	FB_AlarmCodeManager : FB_AlarmCodeManager ; 
	KK				: BYTE;		// For Loop 
	bComError		: BOOL := TRUE;
	bComWarning 	: BOOL;

	AX_BJHS			: ARRAY[1..10] OF BOOL;
END_VAR
FOR KK := 1 TO 19 DO
	bCOmError := bCOmError AND FB_ModbusRead[KK].ModbusReadAlarm;
	bComWarning := bComWarning OR FB_ModbusRead[KK].ModbusReadAlarm;
END_FOR
bComWarning := bComError OR FB_ModbusWrite[1].ModbusWriteAlarm OR FB_ModbusWrite[2].ModbusWriteAlarm ;

TON_ComAlarm(IN := bComError, PT := T#30S,Q=> MesDataExd.MesData.MesAlarmCom);
TON_ComWarning(IN := bComWarning, PT := T#30S, Q=> MesWarningCom);

// ALARM CODE //
	FB_AlarmCodeManager(
		bAlarm1			:= FALSE,												//
		bAlarm2			:= FALSE,                                               //
		bAlarm3			:= FALSE,                                               //
		bAlarm4			:= FALSE,                                               //
		bAlarm5			:= FALSE,												//
		bAlarm6			:= FALSE,												// 
		bAlarm7			:= FALSE,												//
		bAlarm8			:= FALSE,												// 
		bAlarm9			:= FALSE,												//
		bAlarm10		:= FALSE,                                               //
		bAlarm11		:= FALSE,                                               //
		bAlarm12		:= FALSE,                                               //
		bAlarm13		:= FALSE,                                               //
		bAlarm14		:= FALSE,                                               //
		bAlarm15		:= MesDataExd.MesData.MesAlarmCom, 						// No communication frames for the past 30 seconds 					 			#COM
		wAlarmCode		=> MesDataExd.MesData.MesAlarmCode);					

// WARNING CODE //
	FB_AlarmCodeManager(
 		bAlarm1			:= MesWarningCom, 										// A frame failed for the last 30s 												#COM
		bAlarm2			:= FALSE,                                               //
		bAlarm3			:= NOT MesDataExd.MesData.MesCP_Read, 	  				// No permission to read from SCADA
		bAlarm4			:= MesDataExd.ParamID_PMode <> 0,						// INV active power setpoint is not MPPT  										#Equipment
		bAlarm5			:= NOT MesDataExd.MesData.MesCP_Write,					// No permission to write from SCADA							
		bAlarm6			:= FALSE,                                               //
		bAlarm7			:= FALSE,                                               //
		bAlarm8			:= FALSE,												//
		bAlarm9			:= IN_SetptPlimit_Local < MesDataExd.MesData.ParamPn,  	// INV local active power setpoint is under nominal active power 
		bAlarm10		:= NOT RS_StartStop_Local.Q1,       					// Local Stop Command 
		bAlarm11		:= FALSE,						 						// 
		bAlarm12		:= FALSE, 												//
		bAlarm13		:= FALSE,												// 
		bAlarm14		:= FALSE,												// 
		bAlarm15		:= FALSE, 												//
		wAlarmCode		=> MesDataExd.MesData.MesWarningCode);	

// EVENT CODE //
	FB_AlarmCodeManager(
		bAlarm1			:= MesDataExd.MesStateStart_Bbox,                       // Start OK from Bbox
		bAlarm2			:= NOT MesDataExd.MesStateStart_Bbox,                   // Start NOK from Bbox
		bAlarm3			:= MesDataExd.MesStateStart_Freq,                       // Start OK from Freq
		bAlarm4			:= NOT MesDataExd.MesStateStart_Freq,					// Start NOK from Freq
		bAlarm5			:= MesDataExd.MesStateStart_MVCells,                    // Start OK from MV Cells
		bAlarm6			:= NOT MesDataExd.MesStateStart_MVCells,                // Start NOK from MV Cells
		bAlarm7			:= MesDataExd.MesStateStart_P,                          // Start OK from P
		bAlarm8			:= NOT MesDataExd.MesStateStart_P,                      // Start NOK from P
		bAlarm9			:= MesDataExd.MesStateStart_Vdc,                        // Start OK from Vdc
		bAlarm10		:= NOT MesDataExd.MesStateStart_Vdc,                    // Start NOK from Vdc
		bAlarm11		:= NOT RS_StartStop.Q1, 								// Stop command for INV 
		bAlarm12		:= MesDataExd.MesData.MesState_INV = 0,  				// Power Up
		bAlarm13		:= MesDataExd.MesData.MesState_INV = 1,  				// Init
		bAlarm14		:= MesDataExd.MesData.MesState_INV = 2,  				// Off
		bAlarm15		:= MesDataExd.MesData.MesState_INV = 3,  				// Standby DC
		wAlarmCode		=>  MesDataExd.MesData.MesEventCode);
// EVENT CODE //
	FB_AlarmCodeManager(
		bAlarm1			:= MesDataExd.MesData.MesState_INV = 4,  				// Precharge DC
		bAlarm2			:= MesDataExd.MesData.MesState_INV = 5,  				// Softcharge DC
		bAlarm3			:= MesDataExd.MesData.MesState_INV = 6,  				// Ready DC
		bAlarm4			:= MesDataExd.MesData.MesState_INV = 7,  				// Standby AC
		bAlarm5			:= MesDataExd.MesData.MesState_INV = 8,  				// Blackstard
		bAlarm6			:= MesDataExd.MesData.MesState_INV = 9,  				// Ready
		bAlarm7			:= MesDataExd.MesData.MesState_INV = 10,  				// Wait
		bAlarm8			:= MesDataExd.MesData.MesState_INV = 11,  				// Pre ON
		bAlarm9			:= MesDataExd.MesData.MesState_INV = 12,  				// ON
		bAlarm10		:= MesDataExd.MesData.MesState_INV = 13,  				// Stop
		bAlarm11		:= MesDataExd.MesData.MesState_INV = 14,  				// Ready AC
		bAlarm12		:= MesDataExd.MesData.MesState_INV = 15,  				// Diagnostic AC
		bAlarm13		:= MesDataExd.MesData.MesState_INV = 16,  				// Discharge
		bAlarm14		:= MesDataExd.MesData.MesState_INV = 17,  				// Fault
		bAlarm15		:= FALSE,												// 		
		wAlarmCode		=>  MesDataExd.MesEventCode2);

FOR KK := 1 TO CstNbPowerCol_INV_G DO
	FB_AlarmCodeManager(
		bAlarm1			:= MesDataExd.AX_PowerCol[KK].MesState = 0 , // Invalid
		bAlarm2			:= MesDataExd.AX_PowerCol[KK].MesState = 1 , // Stop 
		bAlarm3			:= MesDataExd.AX_PowerCol[KK].MesState = 2 , // Softcharge
		bAlarm4			:= MesDataExd.AX_PowerCol[KK].MesState = 3 , // Ready 
		bAlarm5			:= FALSE,												// 	
		bAlarm6			:= MesDataExd.AX_PowerCol[KK].MesState = 5 , // Pre Run
		bAlarm7			:= MesDataExd.AX_PowerCol[KK].MesState = 6 , // Run
		bAlarm8			:= MesDataExd.AX_PowerCol[KK].MesState = 7 , // Discharge 
		bAlarm9			:= FALSE,												// 	
		bAlarm10		:= FALSE,												// 	
		bAlarm11		:= MesDataExd.AX_PowerCol[KK].MesState = 10, // Wait Over-Current 
		bAlarm12		:= MesDataExd.AX_PowerCol[KK].MesState = 11, // Wait Under-Voltage 
		bAlarm13		:= MesDataExd.AX_PowerCol[KK].MesState = 12, // Over-Current Wait DSP 
		bAlarm14		:= MesDataExd.AX_PowerCol[KK].MesState = 13, // Under-VDC Wait DSP 
		bAlarm15		:= MesDataExd.AX_PowerCol[KK].MesState = 14, // Unbalance VDC Wait DSP 
		wAlarmCode		=>  MesDataExd.AX_PowerCol[KK].MesData.MesEventCode);
	
END_FOR















		
(*
	FB_AlarmCodeManager(
		bAlarm0			:= FALSE, 			// MPPT
		bAlarm1			:= FALSE, 			// Id : Current close loop
		bAlarm2			:= FALSE, 			// P : Power close loop
		bAlarm3			:= FALSE, 			// Vdc : voltage close loop
		bAlarm4			:= FALSE, 			// HT
		bAlarm5			:= FALSE, 			// STAT
		bAlarm6			:= FALSE, 			// R
		bAlarm7			:= FALSE, 			// Night : voltage dc night
		bAlarm8			:= FALSE, 			// 
		bAlarm9			:= FALSE, 			// 
		bAlarm10		:= FALSE, 			// 
		bAlarm11		:= FALSE,			// 
		bAlarm12		:= FALSE,			// 
		bAlarm13		:= FALSE,			// 
		bAlarm14		:= FALSE,			// 
		bAlarm15		:= FALSE,			// 		
		wAlarmCode		=>  MesDataExd.MesStatusCurtail_P);

	FB_AlarmCodeManager(
		bAlarm0			:= FALSE, 			// CosPhi
		bAlarm1			:= FALSE, 			// Iq : Current close loop
		bAlarm2			:= FALSE, 			// Q : Power cose loop
		bAlarm3			:= FALSE, 			// QV : QV Curve
		bAlarm4			:= FALSE, 			// HT
		bAlarm5			:= FALSE, 			// R
		bAlarm6			:= FALSE, 			// 
		bAlarm7			:= FALSE, 			// 
		bAlarm8			:= FALSE, 			// 
		bAlarm9			:= FALSE, 			// 
		bAlarm10		:= FALSE, 			// 
		bAlarm11		:= FALSE,			// 
		bAlarm12		:= FALSE,			// 
		bAlarm13		:= FALSE,			// 
		bAlarm14		:= FALSE,			// 
		bAlarm15		:= FALSE,			// 		
		wAlarmCode		=>  MesDataExd.MesStatusCurtail_Q);

	FB_AlarmCodeManager(
		bAlarm0			:= FALSE, 			// Enable Module 1
		bAlarm1			:= FALSE, 			// Lock Module 1
		bAlarm2			:= FALSE, 			// Enable Module 2
		bAlarm3			:= FALSE, 			// Lock Module 2
		bAlarm4			:= FALSE, 			// Enable Module 3
		bAlarm5			:= FALSE, 			// Lock Module 3
		bAlarm6			:= FALSE, 			// Enable Module 4
		bAlarm7			:= FALSE, 			// Lock Module 4
		bAlarm8			:= FALSE, 			// Enable Module 5
		bAlarm9			:= FALSE, 			// Lock Module 5
		bAlarm10		:= FALSE, 			// Enable Module 6
		bAlarm11		:= FALSE,			// Lock Module 6
		bAlarm12		:= FALSE,			// Enable Module 7
		bAlarm13		:= FALSE,			// Lock Module 7
		bAlarm14		:= FALSE,			// Enable Module 8
		bAlarm15		:= FALSE,			// Lock Module 8
		wAlarmCode		=>  MesDataExd.MesState_Module);

	FB_AlarmCodeManager(
		bAlarm0			:= FALSE, 			// Enable Module 1
		bAlarm1			:= FALSE, 			// Lock Module 1
		bAlarm2			:= FALSE, 			// Enable Module 2
		bAlarm3			:= FALSE, 			// Lock Module 2
		bAlarm4			:= FALSE, 			// Enable Module 3
		bAlarm5			:= FALSE, 			// Lock Module 3
		bAlarm6			:= FALSE, 			// Enable Module 4
		bAlarm7			:= FALSE, 			// Lock Module 4
		bAlarm8			:= FALSE, 			// Enable Module 5
		bAlarm9			:= FALSE, 			// Lock Module 5
		bAlarm10		:= FALSE, 			// Enable Module 6
		bAlarm11		:= FALSE,			// Lock Module 6
		bAlarm12		:= FALSE,			// Enable Module 7
		bAlarm13		:= FALSE,			// Lock Module 7
		bAlarm14		:= FALSE,			// Enable Module 8
		bAlarm15		:= FALSE,			// Lock Module 8
		wAlarmCode		=>  MesDataExd.MesData.MesSate_INV);
		
	FB_AlarmCodeManager(
		bAlarm0			:= FALSE, 			// Stopped
		bAlarm1			:= FALSE, 			// MPPT
		bAlarm2			:= FALSE, 			// Sleeping
		bAlarm3			:= FALSE, 			// Starting
		bAlarm4			:= FALSE, 			// Throttled
		bAlarm5			:= FALSE, 			// Shutting Down
		bAlarm6			:= FALSE, 			// Fault
		bAlarm7			:= FALSE, 			// Standby
		bAlarm8			:= FALSE, 			// 
		bAlarm9			:= FALSE, 			// 
		bAlarm10		:= FALSE, 			// 
		bAlarm11		:= FALSE,			// 
		bAlarm12		:= FALSE,			// 
		bAlarm13		:= FALSE,			// 
		bAlarm14		:= FALSE,			// 
		bAlarm15		:= FALSE,			// 		
		wAlarmCode		=>  MesDataExd.MesData.MesState);		
		
		
*)
END_METHOD

METHOD M_CP
//////////////////
//  Emulator
/////////////////

VAR 
	// Method local variables (reinitialized at each cycle) 
	
END_VAR


SUPER^.M_CP() ; 




Trig_Cmd_Read(CLK:=IN_CmdToggleRead);
Trig_Cmd_Write(CLK:=IN_CmdToggleWrite);
	
IF Trig_Cmd_Read.Q THEN
	IN_CmdToggleRead := FALSE;
	MesDataExd.MesData.MesCP_Read := NOT MesDataExd.MesData.MesCP_Read;
END_IF


IF Trig_Cmd_Write.Q THEN
	IN_CmdToggleWrite := FALSE;
	MesDataExd.MesData.MesCP_Write := NOT MesDataExd.MesData.MesCP_Write;
END_IF
END_METHOD

{attribute 'object_name' := 'M_Curtail'}
METHOD M_Curtail
//////////////////
// Write Curtail Command through modbus to PV inverters.  
//////////////////
VAR 
	// Method local variables (reinitialized at each cycle) 

	MW					: FB_MergeWordsToFloat;
	MW_1				: FB_SplitFloatToWords;
	AX_ADR_MB			: ARRAY[1..3] OF  WORD := [40553, 40558, 40551];
	AX_QTY_MB			: ARRAY[1..3] OF  BYTE := [1, 1, 1];
	
	InvSetptP_temp		: REAL;
	InvSetptQ_temp		: REAL;

	KK: INT;
END_VAR
SUPER^.M_Curtail() ; 

// MODBUS VARIABLE FORMATING //
// Setpoints //
FB_ModbusWrite[1](WriteCmd := FALSE);
FB_ModbusWrite[2](WriteCmd := FALSE);
//FB_ModbusWrite[3](WriteCmd := FALSE);
//FB_ModbusWrite[4](WriteCmd := FALSE);

InvSetptP_temp	:= 10000*IN_SetptPlimit / MesDataExd.MesData.ParamPn; 
InvSetptQ_temp	:= 10000*IN_SetptQ / MesDataExd.MesData.ParamQn; 

MesDataExd.MesData.OUT_SetptPLimit :=  IN_SetptPlimit; 
MesDataExd.MesData.OUT_SetptQ :=  IN_SetptQ; 
	
//IF A1_PP.ParamTanPhiCtrl OR A1_SUBMV.A1_GRID.MesDataExd.OUT_CmdQReg THEN	
//	MesBlockWrite4_Temp[1] := REAL_TO_WORD(InvSetptP_temp);
//	MesBlockWrite4_Temp[6] := REAL_TO_WORD(InvSetptQ_temp);
//ELSE
//	MesBlockWrite4_Temp[1] := REAL_TO_WORD(InvSetptP_temp);	
//	MesBlockWrite4_Temp[6]:= 16#0000;
//END_IF
		
// Regulation mode
// MesBlockWrite5_Temp[1] := INT_TO_WORD(0);
//MesBlockWrite5_Temp[2] := INT_TO_WORD(1);
	
// Send regulation modes
//			FB_ModbusWrite[3]
//		(
//			pSrcAddr := ADR (MesBlockWrite5_Temp[1]),
//			sIPAddr := ParamIPAddress,
//			tTimeout := ParamTimeout,
//			nMBAddr := AX_ADR_MB[3],
//			nTCPport := ParamTCPPort,
//			cbLength := SIZEOF(MesBlockWrite5_Temp[1]),
//			nQuantity := AX_QTY_MB[3],
//			nUnitID := ParamUnitID,
//			WriteCmd := ClockWrite AND MesData.MesCP_Write  ,
//			Reset := CmdClearFault_G OR IN_CmdReset_L,
//			ErrorId => AX_ModbusWriteAlarmId[3],
//			ModbusWriteAlarm => AX_ModbusWriteAlarm[3]
//		);	
//			FB_ModbusWrite[4]
//		(
//			pSrcAddr := ADR (MesBlockWrite5_Temp[2]),
//			sIPAddr := ParamIPAddress,
//			tTimeout := ParamTimeout,
//			nMBAddr := AX_ADR_MB[3]+1,
//			nTCPport := ParamTCPPort,
//			cbLength := SIZEOF(MesBlockWrite5_Temp[2]),
//			nQuantity := AX_QTY_MB[3],
//			nUnitID := ParamUnitID,
//			WriteCmd := ClockWrite AND MesData.MesCP_Write  ,
//			Reset := CmdClearFault_G OR IN_CmdReset_L,
//			ErrorId => AX_ModbusWriteAlarmId[4],
//			ModbusWriteAlarm => AX_ModbusWriteAlarm[4]
//		);		
//	FB_ModbusWrite[1]
//(
//	pSrcAddr := ADR (MesBlockWrite4_Temp[1]),
//	sIPAddr := ParamIPAddress,
//	tTimeout := ParamTimeout,
//	nMBAddr := AX_ADR_MB[1],
//	nTCPport := ParamTCPPort,
//	cbLength := SIZEOF(MesBlockWrite4_Temp[1]),
//	nQuantity := AX_QTY_MB[1],
//	nUnitID := ParamUnitID,
//	WriteCmd := ClockWrite AND MesDataExd.MesData.MesCP_Write  ,
//	Reset := CmdClearFault_G OR IN_CmdReset_L,
//	ErrorId => AX_ModbusWriteAlarmId[1],
//	ModbusWriteAlarm => AX_ModbusWriteAlarm[1]
//);
//
//	FB_ModbusWrite[2]
//(
//	pSrcAddr := ADR (MesBlockWrite4_Temp[6]),
//	sIPAddr := ParamIPAddress,
//	tTimeout := ParamTimeout,
//	nMBAddr := AX_ADR_MB[2],
//	nTCPport := ParamTCPPort,
//	cbLength := SIZEOF(MesBlockWrite4_Temp[6]),
//	nQuantity := AX_QTY_MB[2],
//	nUnitID := ParamUnitID,
//	WriteCmd := ClockWrite AND MesDataExd.MesData.MesCP_Write  ,
//	Reset := CmdClearFault_G OR IN_CmdReset_L,
//	ErrorId => AX_ModbusWriteAlarmId[2],
//	ModbusWriteAlarm => AX_ModbusWriteAlarm[2]
//);
END_METHOD

METHOD M_Evaluate
VAR
	KK	: UINT ;

END_VAR
MesDataExd.MesPAvailable	:= 0;

FOR KK:= 1 TO CstNbDcModule_INV_G DO 												
	MesDataExd.MesPAvailable:= MesDataExd.MesPAvailable + MesDataExd.AX_DcModule[KK].MesPdc;
END_FOR 



MesDataExd.MesP_LV				:=	MesDataExd.MesData.MesP;
MesDataExd.MesQ_LV				:=	MesDataExd.MesData.MesQ;
MesDataExd.MesS_LV				:=	MesDataExd.MesData.MesS;
END_METHOD

METHOD M_Execute
//////////////////
//  Method Calls 
/////////////////

VAR 
	// Method local variables (reinitialized at each cycle) 

END_VAR
IF  bInit THEN
	M_Init();
	bInit:= FALSE ; 
ELSIF CmdInit_G THEN 
	bInit:= TRUE ;
END_IF

SUPER^.M_Execute(); 

M_Evaluate();
M_AlarmManagement();
END_METHOD

METHOD M_Init

VAR
	bCompleted 			: BOOL := FALSE;
	AX_ADR_MB			: WORD := 44253; 
END_VAR
//MesDataExd.MesData.ParamPn := 3800;
IN_SetptPlimit_Local := MesDataExd.MesData.ParamPn;

// Watchdog timer start
Watchdog_CP_Write := TRUE;

// Stop the PPC/INV watchdog timer
FB_ModbusWrite[5](WriteCmd := FALSE);
FB_ModbusWrite[6](WriteCmd := FALSE);

	// Reset refs time / Home P ref / Home Q ref
	MesBlockWrite6_Temp    := REAL_TO_WORD(0);
	MesBlockWrite7_Temp[1] := REAL_TO_WORD(ParamPref_NoCom*100);
	MesBlockWrite7_Temp[2] := REAL_TO_WORD(ParamQref_NoCom*100);
	
	FB_ModbusWrite[5]
	(
		pSrcAddr := ADR (MesBlockWrite6_Temp),
		sIPAddr := ParamIPAddress,
		tTimeout := ParamTimeout,
		nMBAddr := AX_ADR_MB,
		nTCPport := ParamTCPPort,
		cbLength := SIZEOF(MesBlockWrite6_Temp),
		nQuantity := 1,
		nUnitID := ParamUnitID,
		WriteCmd := StartStop_RTrig.Q AND MesDataExd.MesData.MesCP_Write,
		Reset := CmdClearFault_G,
		ErrorId => AX_ModbusWriteAlarmId[5],
		ModbusWriteAlarm => AX_ModbusWriteAlarm[5]
	);
	
		FB_ModbusWrite[6]
	(
		pSrcAddr := ADR (MesBlockWrite7_Temp),
		sIPAddr := ParamIPAddress,
		tTimeout := ParamTimeout,
		nMBAddr := (AX_ADR_MB + 2),
		nTCPport := ParamTCPPort,
		cbLength := SIZEOF(MesBlockWrite7_Temp),
		nQuantity := 2,
		nUnitID := ParamUnitID,
		WriteCmd := StartStop_RTrig.Q AND MesDataExd.MesData.MesCP_Write,
		Reset := CmdClearFault_G,
		ErrorId => AX_ModbusWriteAlarmId[6],
		ModbusWriteAlarm => AX_ModbusWriteAlarm[6]
	);
END_METHOD

{attribute 'object_name' := 'M_Read'}
METHOD M_Read
//////////
// Read Method for PE SKID HEMK : Modbus reading
//////////
VAR
	// Method local variables (reinitialized at each cycle) 
	MW_Float			: FB_MergeWordsToFloat;
	MW_REAL				: FB_MergeWordsToDint;
	MW_UInt				: FB_MergeWordsToUint;
	
	MesUdc				: REAL;
	Mesfreq				: UINT;
	
	KK					: BYTE;						 // Index to loop over modbus blocks 	
	JJ					: BYTE;
	LL 					: UINT;
	NbModules			: UINT;
	
	test_uint : UINT;
	
END_VAR
// CP-Read / Write 

IF MesDataExd.MesData.MesCP_Read THEN		

	// MODBUS REQUEST//
		//Energy daily and total per PowerModule
		FB_ModbusRead[1]
		(
			nTCPPort		:= ParamTcpPort,
			ClockRead		:= MesDataExd.MesData.MesCP_Read AND ClockRead, 
			Reset			:= CmdClearFault_G OR IN_CmdReset_L,
			sIPAddr			:=ParamIPAddress ,
			nUnitID			:= 1, 
			tTimeout		:= ParamTimeout,
			nQuantity		:= AX_QTY_MB[1] , 
			nMBAddr			:= AX_ADR_MB[1] , 
			cbLength		:= SIZEOF(MesBlock_Temp_1) , 
			pDestAddr		:= ADR(MesBlock_Temp_1) , 
			ModbusReadAlarm	=>AX_ModbusReadAlarm[1] , 
			ErrorId			=> AX_ModbusReadAlarmId[1]
		);
			
		//DC Switch status
		FB_ModbusRead[2]
		(
			nTCPPort		:= ParamTcpPort,
			ClockRead		:= MesDataExd.MesData.MesCP_Read AND ClockRead, 
			Reset			:= CmdClearFault_G OR IN_CmdReset_L,
			sIPAddr			:=ParamIPAddress , 
			nUnitID			:= 1, 
			tTimeout		:= ParamTimeout,
			nQuantity		:= AX_QTY_MB[2] , 
			nMBAddr			:= AX_ADR_MB[2] , 
			cbLength		:= SIZEOF(MesBlock_Temp_2) , 
			pDestAddr		:= ADR(MesBlock_Temp_2) , 
			ModbusReadAlarm	=>AX_ModbusReadAlarm[2] , 
			ErrorId			=> AX_ModbusReadAlarmId[2]
		);
		
		// Statuses and P / Q control
		FB_ModbusRead[3]
		(
			nTCPPort		:= ParamTcpPort,
			ClockRead		:= MesDataExd.MesData.MesCP_Read AND ClockRead, 
			Reset			:= CmdClearFault_G OR IN_CmdReset_L,
			sIPAddr			:=ParamIPAddress , 
			nUnitID			:= 1, 
			tTimeout		:= ParamTimeout,
			nQuantity		:= AX_QTY_MB[3] , 
			nMBAddr			:= AX_ADR_MB[3] , 
			cbLength		:= SIZEOF(MesBlock_Temp_3) , 
			pDestAddr		:= ADR(MesBlock_Temp_3) , 
			ModbusReadAlarm	=>AX_ModbusReadAlarm[3] , 
			ErrorId			=> AX_ModbusReadAlarmId[3]
		);
		
		//DC Modules
		FB_ModbusRead[4]
		(
			nTCPPort		:= ParamTcpPort,
			ClockRead		:= MesDataExd.MesData.MesCP_Read AND ClockRead, 
			Reset			:= CmdClearFault_G OR IN_CmdReset_L,
			sIPAddr			:= ParamIPAddress , 
			nUnitID			:= 1, 
			tTimeout		:= ParamTimeout,
			nQuantity		:= AX_QTY_MB[4], 
			nMBAddr			:= AX_ADR_MB[4], 
			cbLength		:= SIZEOF(MesBlock_Temp_4), 
			pDestAddr		:= ADR(MesBlock_Temp_4), 
			ModbusReadAlarm	=> AX_ModbusReadAlarm[4], 
			ErrorId			=> AX_ModbusReadAlarmId[4]
		);
		
		FB_ModbusRead[5]
		(
			nTCPPort		:= ParamTcpPort,
			ClockRead		:= MesDataExd.MesData.MesCP_Read AND ClockRead, 
			Reset			:= CmdClearFault_G OR IN_CmdReset_L,
			sIPAddr			:= ParamIPAddress , 
			nUnitID			:= 1, 
			tTimeout		:= ParamTimeout,
			nQuantity		:= AX_QTY_MB[5], 
			nMBAddr			:= AX_ADR_MB[5], 
			cbLength		:= SIZEOF(MesBlock_Temp_5), 
			pDestAddr		:= ADR(MesBlock_Temp_5), 
			ModbusReadAlarm	=> AX_ModbusReadAlarm[5], 
			ErrorId			=> AX_ModbusReadAlarmId[5]
		);
		
		FB_ModbusRead[6]
		(
			nTCPPort		:= ParamTcpPort,
			ClockRead		:= MesDataExd.MesData.MesCP_Read AND ClockRead, 
			Reset			:= CmdClearFault_G OR IN_CmdReset_L,
			sIPAddr			:= ParamIPAddress , 
			nUnitID			:= 1, 
			tTimeout		:= ParamTimeout,
			nQuantity		:= AX_QTY_MB[6], 
			nMBAddr			:= AX_ADR_MB[6], 
			cbLength		:= SIZEOF(MesBlock_Temp_6), 
			pDestAddr		:= ADR(MesBlock_Temp_6), 
			ModbusReadAlarm	=> AX_ModbusReadAlarm[6], 
			ErrorId			=> AX_ModbusReadAlarmId[6]
		);
		
		FB_ModbusRead[7]
		(
			nTCPPort		:= ParamTcpPort,
			ClockRead		:= MesDataExd.MesData.MesCP_Read AND ClockRead, 
			Reset			:= CmdClearFault_G OR IN_CmdReset_L,
			sIPAddr			:= ParamIPAddress , 
			nUnitID			:= 1, 
			tTimeout		:= ParamTimeout,
			nQuantity		:= AX_QTY_MB[7], 
			nMBAddr			:= AX_ADR_MB[7], 
			cbLength		:= SIZEOF(MesBlock_Temp_7), 
			pDestAddr		:= ADR(MesBlock_Temp_7), 
			ModbusReadAlarm	=> AX_ModbusReadAlarm[7], 
			ErrorId			=> AX_ModbusReadAlarmId[7]
		);
		//Power Commands
		FOR KK:= 1 TO  CstNbPowerCol_INV_G DO 
			FB_ModbusRead[7 + KK]
			(
					nTCPPort		:= ParamTcpPort,
					ClockRead		:= MesDataExd.MesData.MesCP_Read AND ClockRead, 
					Reset			:= CmdClearFault_G OR IN_CmdReset_L,
					sIPAddr			:=ParamIPAddress , 
					nUnitID			:= 1, 
					tTimeout		:= ParamTimeout,
					nQuantity		:= AX_QTY_MB[8] , 
					nMBAddr			:= AX_ADR_MB[8] + 35*(KK-1) ,  
					cbLength		:= SIZEOF(MesBlock_Temp_8[KK]) , 
					pDestAddr		:= ADR(MesBlock_Temp_8[KK]) , 
					ModbusReadAlarm	=>AX_ModbusReadAlarm[7+KK] , 
					ErrorId			=> AX_ModbusReadAlarmId[7+KK]
			);
		END_FOR
		FB_ModbusRead[20]
		(
				nTCPPort		:= ParamTcpPort,
				ClockRead		:= MesDataExd.MesData.MesCP_Read AND ClockRead, 
				Reset			:= CmdClearFault_G OR IN_CmdReset_L,
				sIPAddr			:=ParamIPAddress , 
				nUnitID			:= 1, 
				tTimeout		:= ParamTimeout,
				nQuantity		:= 2, 
				nMBAddr			:= 2313 ,  
				cbLength		:= SIZEOF(MesBlock_Temp_9) , 
				pDestAddr		:= ADR(MesBlock_Temp_9) , 
				ModbusReadAlarm	=>AX_ModbusReadAlarm[20] , 
				ErrorId			=> AX_ModbusReadAlarmId[20]
		);		
	// Block reading
		// Block1
			MW_UInt(WORD_STRONG:= MesBlock_Temp_1[ 1],WORD_WEAK:=MesBlock_Temp_1[ 2], VAR_OUT:=MesDataExd.MesAcDay);
			MW_UInt(WORD_STRONG:= MesBlock_Temp_1[ 9],WORD_WEAK:=MesBlock_Temp_1[ 10], VAR_OUT:=MesDataExd.MesAcTot);   
		
		// Block2
			MesDataExd.AX_DcModule[1].MesClosed_DcSwitch := MesBlock_Temp_2[1] = 1;
			MesDataExd.AX_DcModule[2].MesClosed_DcSwitch := MesBlock_Temp_2[2] = 1;
			MesDataExd.AX_DcModule[3].MesClosed_DcSwitch := MesBlock_Temp_2[3] = 1;
			MesDataExd.AX_DcModule[4].MesClosed_DcSwitch := MesBlock_Temp_2[4] = 1;
			MesDataExd.AX_DcModule[1].MesChargedSpring := MesBlock_Temp_2[5] = 1;
			MesDataExd.AX_DcModule[2].MesChargedSpring := MesBlock_Temp_2[6] = 1;
			MesDataExd.AX_DcModule[3].MesChargedSpring := MesBlock_Temp_2[7] = 1;
			MesDataExd.AX_DcModule[4].MesChargedSpring := MesBlock_Temp_2[8] = 1;
			
			
		// Block3
			MesDataExd.MesIDFault 					:= WORD_TO_UINT(MesBlock_Temp_3[1]);
			MesDataExd.MesIDLastFaultedPowerCol 	:= WORD_TO_UINT(MesBlock_Temp_3[2]);
			MesDataExd.MesIDWarning 				:= WORD_TO_UINT(MesBlock_Temp_3[3]);
			MesDataExd.MesData.MesState_INV			:= WORD_TO_UINT(MesBlock_Temp_3[4]);
			MesDataExd.MesStateStart_Freq			:= WORD_TO_BOOL(MesBlock_Temp_3[41]);
			MesDataExd.MesStateStart_Vdc		    := WORD_TO_BOOL(MesBlock_Temp_3[42]);
			MesDataExd.MesStateStart_MVCells	    := WORD_TO_BOOL(MesBlock_Temp_3[43]);
			MesDataExd.MesStateStart_P			    := WORD_TO_BOOL(MesBlock_Temp_3[44]);
			MesDataExd.MesStateStart_Bbox		    := WORD_TO_BOOL(MesBlock_Temp_3[45]);
			MW_REAL(WORD_STRONG:= MesBlock_Temp_3[ 61], SIGNED:=FALSE, FIX:=2 , SIZE:=1, VAR_OUT:=MesDataExd.MesSetptP); // En réalité Plimit 
			MW_REAL(WORD_STRONG:= MesBlock_Temp_3[ 62], SIGNED:=FALSE, FIX:=2 , SIZE:=1, VAR_OUT:=MesDataExd.MesSetptQ); // En réalité Qlimit
 			MW_REAL(WORD_STRONG:= MesBlock_Temp_3[ 66], SIGNED:=FALSE, FIX:=2 , SIZE:=1, VAR_OUT:=MesDataExd.MesPn);
			MW_REAL(WORD_STRONG:= MesBlock_Temp_3[ 72], SIGNED:=FALSE, FIX:=-1 , SIZE:=1, VAR_OUT:=MesDataExd.MesData.MesInsuResistor);
			MW_REAL(WORD_STRONG:= MesBlock_Temp_3[ 101], SIGNED:=TRUE, FIX:=0 , SIZE:=1, VAR_OUT:=MesDataExd.MesTemp_Internal);
			MW_REAL(WORD_STRONG:= MesBlock_Temp_3[ 109], SIGNED:=TRUE, FIX:=0 , SIZE:=1, VAR_OUT:=MesDataExd.MesData.MesTemp);
			MesDataExd.MesStatusCurtail_P			:= MesBlock_Temp_3[112]; // correction KBT : test, valeur semble plus cohérente
			MesDataExd.MesStatusCurtail_Q			:= MesBlock_Temp_3[114];
			MW_REAL(WORD_STRONG:= MesBlock_Temp_3[ 119], SIGNED:=FALSE, FIX:=1 , SIZE:=1, VAR_OUT:=MesDataExd.MesDeratingGlobal);
		
		// Block 4
			MW_REAL(WORD_STRONG:= MesBlock_Temp_4[  1], SIGNED:=TRUE, FIX:=0 , SIZE:=1, VAR_OUT:=MesDataExd.AX_DcModule[1].MesPdc);
			MW_REAL(WORD_STRONG:= MesBlock_Temp_4[  2], SIGNED:=TRUE, FIX:=0 , SIZE:=1, VAR_OUT:=MesDataExd.AX_DcModule[2].MesPdc);
			MW_REAL(WORD_STRONG:= MesBlock_Temp_4[  3], SIGNED:=TRUE, FIX:=0 , SIZE:=1, VAR_OUT:=MesDataExd.AX_DcModule[3].MesPdc);
			MW_REAL(WORD_STRONG:= MesBlock_Temp_4[  4], SIGNED:=TRUE, FIX:=0 , SIZE:=1, VAR_OUT:=MesDataExd.AX_DcModule[4].MesPdc);
			MW_REAL(WORD_STRONG:= MesBlock_Temp_4[  5], SIGNED:=TRUE, FIX:=0 , SIZE:=1, VAR_OUT:=MesDataExd.AX_DcModule[1].MesIdc);
			MW_REAL(WORD_STRONG:= MesBlock_Temp_4[  6], SIGNED:=TRUE, FIX:=0 , SIZE:=1, VAR_OUT:=MesDataExd.AX_DcModule[2].MesIdc);
			MW_REAL(WORD_STRONG:= MesBlock_Temp_4[  7], SIGNED:=TRUE, FIX:=0 , SIZE:=1, VAR_OUT:=MesDataExd.AX_DcModule[3].MesIdc);
			MW_REAL(WORD_STRONG:= MesBlock_Temp_4[  8], SIGNED:=TRUE, FIX:=0 , SIZE:=1, VAR_OUT:=MesDataExd.AX_DcModule[4].MesIdc);
			MW_REAL(WORD_STRONG:= MesBlock_Temp_4[  9], SIGNED:=TRUE, FIX:=0 , SIZE:=1, VAR_OUT:=MesDataExd.AX_DcModule[1].MesUdc);
			MW_REAL(WORD_STRONG:= MesBlock_Temp_4[ 10], SIGNED:=TRUE, FIX:=0 , SIZE:=1, VAR_OUT:=MesDataExd.AX_DcModule[2].MesUdc);
			MW_REAL(WORD_STRONG:= MesBlock_Temp_4[ 11], SIGNED:=TRUE, FIX:=0 , SIZE:=1, VAR_OUT:=MesDataExd.AX_DcModule[3].MesUdc);
			MW_REAL(WORD_STRONG:= MesBlock_Temp_4[ 12], SIGNED:=TRUE, FIX:=0 , SIZE:=1, VAR_OUT:=MesDataExd.AX_DcModule[4].MesUdc);
		
		// Block 5
			MW_REAL(WORD_STRONG:= MesBlock_Temp_5[  1], SIGNED:=FALSE, FIX:=1 , SIZE:=1, VAR_OUT:=MesDataExd.MesU12);
			MW_REAL(WORD_STRONG:= MesBlock_Temp_5[  2], SIGNED:=FALSE, FIX:=1 , SIZE:=1, VAR_OUT:=MesDataExd.MesU23);
			MW_REAL(WORD_STRONG:= MesBlock_Temp_5[  3], SIGNED:=FALSE, FIX:=1 , SIZE:=1, VAR_OUT:=MesDataExd.MesU31);
			MW_REAL(WORD_STRONG:= MesBlock_Temp_5[  4], SIGNED:=TRUE,  FIX:=1 , SIZE:=1, VAR_OUT:=MesDataExd.MesI1);
			MW_REAL(WORD_STRONG:= MesBlock_Temp_5[  5], SIGNED:=TRUE,  FIX:=1 , SIZE:=1, VAR_OUT:=MesDataExd.MesI2);
			MW_REAL(WORD_STRONG:= MesBlock_Temp_5[  6], SIGNED:=TRUE,  FIX:=1 , SIZE:=1, VAR_OUT:=MesDataExd.MesI3);
//			MW_REAL(WORD_STRONG:= MesBlock_Temp_5[  7], SIGNED:=TRUE,  FIX:=0 , SIZE:=1, VAR_OUT:=MesDataExd.MesData.MesP);
//			MW_REAL(WORD_STRONG:= MesBlock_Temp_5[  8], SIGNED:=TRUE,  FIX:=0 , SIZE:=1, VAR_OUT:=MesDataExd.MesData.MesQ);
//			MW_REAL(WORD_STRONG:= MesBlock_Temp_5[  9], SIGNED:=FALSE, FIX:=0 , SIZE:=1, VAR_OUT:=MesDataExd.MesData.MesS);
//			MW_REAL(WORD_STRONG:= MesBlock_Temp_5[ 10], SIGNED:=TRUE,  FIX:=3 , SIZE:=1, VAR_OUT:=MesDataExd.MesData.MesCosPhi);
			MW_REAL(WORD_STRONG:= MesBlock_Temp_5[ 21], SIGNED:=FALSE, FIX:=1 , SIZE:=1, VAR_OUT:=MesDataExd.MesU12_LV);
			MW_REAL(WORD_STRONG:= MesBlock_Temp_5[ 22], SIGNED:=FALSE, FIX:=1 , SIZE:=1, VAR_OUT:=MesDataExd.MesU23_LV);
			MW_REAL(WORD_STRONG:= MesBlock_Temp_5[ 23], SIGNED:=FALSE, FIX:=1 , SIZE:=1, VAR_OUT:=MesDataExd.MesU31_LV);
			MW_REAL(WORD_STRONG:= MesBlock_Temp_5[ 24], SIGNED:=TRUE,  FIX:=1 , SIZE:=1, VAR_OUT:=MesDataExd.MesI1_LV);
			MW_REAL(WORD_STRONG:= MesBlock_Temp_5[ 25], SIGNED:=TRUE,  FIX:=1 , SIZE:=1, VAR_OUT:=MesDataExd.MesI2_LV);
			MW_REAL(WORD_STRONG:= MesBlock_Temp_5[ 26], SIGNED:=TRUE,  FIX:=1 , SIZE:=1, VAR_OUT:=MesDataExd.MesI3_LV);
			MW_REAL(WORD_STRONG:= MesBlock_Temp_5[ 27], SIGNED:=TRUE,  FIX:=0 , SIZE:=1, VAR_OUT:=MesDataExd.MesData.MesP);
			MW_REAL(WORD_STRONG:= MesBlock_Temp_5[ 28], SIGNED:=TRUE,  FIX:=0 , SIZE:=1, VAR_OUT:=MesDataExd.MesData.MesQ);
			MW_REAL(WORD_STRONG:= MesBlock_Temp_5[ 29], SIGNED:=FALSE, FIX:=0 , SIZE:=1, VAR_OUT:=MesDataExd.MesData.MesS);
			MW_REAL(WORD_STRONG:= MesBlock_Temp_5[ 30], SIGNED:=TRUE,  FIX:=3 , SIZE:=1, VAR_OUT:=MesDataExd.MesData.MesCosPhi);
			MW_REAL(WORD_WEAK:= MesBlock_Temp_5[ 33], WORD_STRONG:= MesBlock_Temp_5[ 32], SIGNED:=TRUE,  FIX:=4 , SIZE:=2, VAR_OUT:=MesDataExd.MesData.MesFreq);

		// Block 6
			MW_REAL(WORD_STRONG:= MesBlock_Temp_6[  1], SIGNED:=TRUE, FIX:=1 , SIZE:=1, VAR_OUT:=MesDataExd.AX_DcModule[1].AX_STR[ 1].MesIdc);
			MW_REAL(WORD_STRONG:= MesBlock_Temp_6[  2], SIGNED:=TRUE, FIX:=1 , SIZE:=1, VAR_OUT:=MesDataExd.AX_DcModule[1].AX_STR[ 2].MesIdc);
			MW_REAL(WORD_STRONG:= MesBlock_Temp_6[  3], SIGNED:=TRUE, FIX:=1 , SIZE:=1, VAR_OUT:=MesDataExd.AX_DcModule[1].AX_STR[ 3].MesIdc);
			MW_REAL(WORD_STRONG:= MesBlock_Temp_6[  4], SIGNED:=TRUE, FIX:=1 , SIZE:=1, VAR_OUT:=MesDataExd.AX_DcModule[1].AX_STR[ 4].MesIdc);
			MW_REAL(WORD_STRONG:= MesBlock_Temp_6[  5], SIGNED:=TRUE, FIX:=1 , SIZE:=1, VAR_OUT:=MesDataExd.AX_DcModule[1].AX_STR[ 5].MesIdc);
			MW_REAL(WORD_STRONG:= MesBlock_Temp_6[  6], SIGNED:=TRUE, FIX:=1 , SIZE:=1, VAR_OUT:=MesDataExd.AX_DcModule[1].AX_STR[ 6].MesIdc);
			MW_REAL(WORD_STRONG:= MesBlock_Temp_6[  7], SIGNED:=TRUE, FIX:=1 , SIZE:=1, VAR_OUT:=MesDataExd.AX_DcModule[1].AX_STR[ 7].MesIdc);
			MW_REAL(WORD_STRONG:= MesBlock_Temp_6[  8], SIGNED:=TRUE, FIX:=1 , SIZE:=1, VAR_OUT:=MesDataExd.AX_DcModule[1].AX_STR[ 8].MesIdc);
			MW_REAL(WORD_STRONG:= MesBlock_Temp_6[  9], SIGNED:=TRUE, FIX:=1 , SIZE:=1, VAR_OUT:=MesDataExd.AX_DcModule[1].AX_STR[ 9].MesIdc);
			MW_REAL(WORD_STRONG:= MesBlock_Temp_6[ 10], SIGNED:=TRUE, FIX:=1 , SIZE:=1, VAR_OUT:=MesDataExd.AX_DcModule[1].AX_STR[10].MesIdc);
			MW_REAL(WORD_STRONG:= MesBlock_Temp_6[ 11], SIGNED:=TRUE, FIX:=1 , SIZE:=1, VAR_OUT:=MesDataExd.AX_DcModule[2].AX_STR[ 1].MesIdc);
			MW_REAL(WORD_STRONG:= MesBlock_Temp_6[ 12], SIGNED:=TRUE, FIX:=1 , SIZE:=1, VAR_OUT:=MesDataExd.AX_DcModule[2].AX_STR[ 2].MesIdc);
			MW_REAL(WORD_STRONG:= MesBlock_Temp_6[ 13], SIGNED:=TRUE, FIX:=1 , SIZE:=1, VAR_OUT:=MesDataExd.AX_DcModule[2].AX_STR[ 3].MesIdc);
			MW_REAL(WORD_STRONG:= MesBlock_Temp_6[ 14], SIGNED:=TRUE, FIX:=1 , SIZE:=1, VAR_OUT:=MesDataExd.AX_DcModule[2].AX_STR[ 4].MesIdc);
			MW_REAL(WORD_STRONG:= MesBlock_Temp_6[ 15], SIGNED:=TRUE, FIX:=1 , SIZE:=1, VAR_OUT:=MesDataExd.AX_DcModule[2].AX_STR[ 5].MesIdc);
			MW_REAL(WORD_STRONG:= MesBlock_Temp_6[ 16], SIGNED:=TRUE, FIX:=1 , SIZE:=1, VAR_OUT:=MesDataExd.AX_DcModule[2].AX_STR[ 6].MesIdc);
			MW_REAL(WORD_STRONG:= MesBlock_Temp_6[ 17], SIGNED:=TRUE, FIX:=1 , SIZE:=1, VAR_OUT:=MesDataExd.AX_DcModule[2].AX_STR[ 7].MesIdc);
			MW_REAL(WORD_STRONG:= MesBlock_Temp_6[ 18], SIGNED:=TRUE, FIX:=1 , SIZE:=1, VAR_OUT:=MesDataExd.AX_DcModule[2].AX_STR[ 8].MesIdc);
			MW_REAL(WORD_STRONG:= MesBlock_Temp_6[ 19], SIGNED:=TRUE, FIX:=1 , SIZE:=1, VAR_OUT:=MesDataExd.AX_DcModule[2].AX_STR[ 9].MesIdc);
			MW_REAL(WORD_STRONG:= MesBlock_Temp_6[ 20], SIGNED:=TRUE, FIX:=1 , SIZE:=1, VAR_OUT:=MesDataExd.AX_DcModule[2].AX_STR[10].MesIdc);
			MW_REAL(WORD_STRONG:= MesBlock_Temp_6[ 21], SIGNED:=TRUE, FIX:=1 , SIZE:=1, VAR_OUT:=MesDataExd.AX_DcModule[3].AX_STR[ 1].MesIdc);
			MW_REAL(WORD_STRONG:= MesBlock_Temp_6[ 22], SIGNED:=TRUE, FIX:=1 , SIZE:=1, VAR_OUT:=MesDataExd.AX_DcModule[3].AX_STR[ 2].MesIdc);
			MW_REAL(WORD_STRONG:= MesBlock_Temp_6[ 23], SIGNED:=TRUE, FIX:=1 , SIZE:=1, VAR_OUT:=MesDataExd.AX_DcModule[3].AX_STR[ 3].MesIdc);
			MW_REAL(WORD_STRONG:= MesBlock_Temp_6[ 24], SIGNED:=TRUE, FIX:=1 , SIZE:=1, VAR_OUT:=MesDataExd.AX_DcModule[3].AX_STR[ 4].MesIdc);
			MW_REAL(WORD_STRONG:= MesBlock_Temp_6[ 25], SIGNED:=TRUE, FIX:=1 , SIZE:=1, VAR_OUT:=MesDataExd.AX_DcModule[3].AX_STR[ 5].MesIdc);
			MW_REAL(WORD_STRONG:= MesBlock_Temp_6[ 26], SIGNED:=TRUE, FIX:=1 , SIZE:=1, VAR_OUT:=MesDataExd.AX_DcModule[3].AX_STR[ 6].MesIdc);
			MW_REAL(WORD_STRONG:= MesBlock_Temp_6[ 27], SIGNED:=TRUE, FIX:=1 , SIZE:=1, VAR_OUT:=MesDataExd.AX_DcModule[3].AX_STR[ 7].MesIdc);
			MW_REAL(WORD_STRONG:= MesBlock_Temp_6[ 28], SIGNED:=TRUE, FIX:=1 , SIZE:=1, VAR_OUT:=MesDataExd.AX_DcModule[3].AX_STR[ 8].MesIdc);
			MW_REAL(WORD_STRONG:= MesBlock_Temp_6[ 29], SIGNED:=TRUE, FIX:=1 , SIZE:=1, VAR_OUT:=MesDataExd.AX_DcModule[3].AX_STR[ 9].MesIdc);
			MW_REAL(WORD_STRONG:= MesBlock_Temp_6[ 30], SIGNED:=TRUE, FIX:=1 , SIZE:=1, VAR_OUT:=MesDataExd.AX_DcModule[3].AX_STR[10].MesIdc);
			MW_REAL(WORD_STRONG:= MesBlock_Temp_6[ 31], SIGNED:=TRUE, FIX:=1 , SIZE:=1, VAR_OUT:=MesDataExd.AX_DcModule[4].AX_STR[ 1].MesIdc);
			MW_REAL(WORD_STRONG:= MesBlock_Temp_6[ 32], SIGNED:=TRUE, FIX:=1 , SIZE:=1, VAR_OUT:=MesDataExd.AX_DcModule[4].AX_STR[ 2].MesIdc);
			MW_REAL(WORD_STRONG:= MesBlock_Temp_6[ 33], SIGNED:=TRUE, FIX:=1 , SIZE:=1, VAR_OUT:=MesDataExd.AX_DcModule[4].AX_STR[ 3].MesIdc);
			MW_REAL(WORD_STRONG:= MesBlock_Temp_6[ 34], SIGNED:=TRUE, FIX:=1 , SIZE:=1, VAR_OUT:=MesDataExd.AX_DcModule[4].AX_STR[ 4].MesIdc);
			MW_REAL(WORD_STRONG:= MesBlock_Temp_6[ 35], SIGNED:=TRUE, FIX:=1 , SIZE:=1, VAR_OUT:=MesDataExd.AX_DcModule[4].AX_STR[ 5].MesIdc);
			MW_REAL(WORD_STRONG:= MesBlock_Temp_6[ 36], SIGNED:=TRUE, FIX:=1 , SIZE:=1, VAR_OUT:=MesDataExd.AX_DcModule[4].AX_STR[ 6].MesIdc);
			MW_REAL(WORD_STRONG:= MesBlock_Temp_6[ 37], SIGNED:=TRUE, FIX:=1 , SIZE:=1, VAR_OUT:=MesDataExd.AX_DcModule[4].AX_STR[ 7].MesIdc);
			MW_REAL(WORD_STRONG:= MesBlock_Temp_6[ 38], SIGNED:=TRUE, FIX:=1 , SIZE:=1, VAR_OUT:=MesDataExd.AX_DcModule[4].AX_STR[ 8].MesIdc);
			MW_REAL(WORD_STRONG:= MesBlock_Temp_6[ 39], SIGNED:=TRUE, FIX:=1 , SIZE:=1, VAR_OUT:=MesDataExd.AX_DcModule[4].AX_STR[ 9].MesIdc);
			MW_REAL(WORD_STRONG:= MesBlock_Temp_6[ 40], SIGNED:=TRUE, FIX:=1 , SIZE:=1, VAR_OUT:=MesDataExd.AX_DcModule[4].AX_STR[10].MesIdc);
		
		//Block 7
			MesDataExd.MesState_Module := MesBlock_Temp_7[1];
			MesDataExd.MesNbRunningModules := WORD_TO_UINT(MesBlock_Temp_7[2]);
			
		//Block 8
		
			FOR KK := 1 TO CstNbPowerCol_INV_G DO
				MesDataExd.AX_PowerCol[KK].MesState := WORD_TO_UINT(MesBlock_Temp_8[KK][1]);
				MW_REAL(WORD_STRONG:= MesBlock_Temp_8[KK][  2], SIGNED:=FALSE, FIX:=1 , SIZE:=1, VAR_OUT:=MesDataExd.AX_PowerCol[KK].MesData.MesI1);
				MW_REAL(WORD_STRONG:= MesBlock_Temp_8[KK][  3], SIGNED:=FALSE, FIX:=1 , SIZE:=1, VAR_OUT:=MesDataExd.AX_PowerCol[KK].MesData.MesI2);
				MW_REAL(WORD_STRONG:= MesBlock_Temp_8[KK][  4], SIGNED:=FALSE, FIX:=1 , SIZE:=1, VAR_OUT:=MesDataExd.AX_PowerCol[KK].MesData.MesI3);
				MW_REAL(WORD_STRONG:= MesBlock_Temp_8[KK][  5], SIGNED:=TRUE,  FIX:=1 , SIZE:=1, VAR_OUT:=MesDataExd.AX_PowerCol[KK].MesData.MesIdc);
				MW_REAL(WORD_STRONG:= MesBlock_Temp_8[KK][  8], SIGNED:=FALSE, FIX:=0 , SIZE:=1, VAR_OUT:=MesDataExd.AX_PowerCol[KK].MesData.MesUdc);
				MW_REAL(WORD_STRONG:= MesBlock_Temp_8[KK][  9], SIGNED:=TRUE,  FIX:=1 , SIZE:=1, VAR_OUT:=MesDataExd.AX_PowerCol[KK].MesData.MesP);
				MW_REAL(WORD_STRONG:= MesBlock_Temp_8[KK][ 10], SIGNED:=TRUE,  FIX:=1 , SIZE:=1, VAR_OUT:=MesDataExd.AX_PowerCol[KK].MesData.MesQ);
				MW_REAL(WORD_STRONG:= MesBlock_Temp_8[KK][ 11], SIGNED:=TRUE,  FIX:=0 , SIZE:=1, VAR_OUT:=MesDataExd.AX_PowerCol[KK].MesTemp);
				MW_REAL(WORD_STRONG:= MesBlock_Temp_8[KK][ 12], SIGNED:=TRUE,  FIX:=2 , SIZE:=1, VAR_OUT:=MesDataExd.AX_PowerCol[KK].MesTempmax);
				MW_REAL(WORD_STRONG:= MesBlock_Temp_8[KK][ 28], SIGNED:=FALSE, FIX:=0 , SIZE:=1, VAR_OUT:=MesDataExd.AX_PowerCol[KK].MesHygro);
				MesUdc := MesUdc + MesDataExd.AX_PowerCol[KK].MesData.MesUdc;
				
				MW_REAL(WORD_STRONG:= MesBlock_Temp_8[KK][ 29], SIGNED:=FALSE, FIX:=0 , SIZE:=1, VAR_OUT:=MesDataExd.AX_PowerCol[KK].MesU12);
				MW_REAL(WORD_STRONG:= MesBlock_Temp_8[KK][ 30], SIGNED:=FALSE, FIX:=0 , SIZE:=1, VAR_OUT:=MesDataExd.AX_PowerCol[KK].MesU23);
				MW_REAL(WORD_STRONG:= MesBlock_Temp_8[KK][ 31], SIGNED:=FALSE, FIX:=0 , SIZE:=1, VAR_OUT:=MesDataExd.AX_PowerCol[KK].MesU31);
				
			END_FOR
	
	MW_UInt(WORD_WEAK:= MesBlock_Temp_9[ 2], WORD_STRONG:= MesBlock_Temp_9[ 1], VAR_OUT:=test_uint);
	
	// MesDataExd.MesData.MesInsuResistor := UINT_TO_REAL(test_uint);
	
	
	
	IF MesDataExd.MesNbRunningModules > 0 THEN
		MesDataExd.MesData.MesUdc := MesUdc/MesDataExd.MesNbRunningModules;		
	END_IF
		
	MesDataExd.MesData.MesPdc					:= MesDataExd.AX_DcModule[1].MesPdc + MesDataExd.AX_DcModule[2].MesPdc + MesDataExd.AX_DcModule[3].MesPdc + MesDataExd.AX_DcModule[4].MesPdc;
	MesDataExd.MesData.MesTemp := 0;
	FOR LL := 1 TO CstNbPowerCol_INV_G DO
		NbModules							:= NbModules + SEL(MesDataExd.AX_PowerCol[LL].MesTemp > 0, 0, 1);
		MesDataExd.MesData.MesTemp			:= MesDataExd.MesData.MesTemp + MesDataExd.AX_PowerCol[LL].MesTemp;
	END_FOR
	MesDataExd.MesData.MesTemp := MesDataExd.MesData.MesTemp/NbModules;

	MesDataExd.MesData.MesI						:= (MesDataExd.MesI1 + MesDataExd.MesI2 + MesDataExd.MesI3) /3;
	MesDataExd.MesData.MesU						:= (MesDataExd.MesU12 + MesDataExd.MesU23 + MesdataExd.MesU31) /3 ;
	MesDataExd.MesData.MesV			    		:= MesDataExd.MesData.MesU/SQRT(3) ; 
	
	                                			
	MesDataExd.MesData.MesAlarmCom  			:= TON_ComAlarm.Q; 
                                    			                                                        	
END_IF
END_METHOD

METHOD M_StartStop
VAR
	KK : UINT;
	AX_ADR_MB			: ARRAY[1..3] OF WORD := [43010, 43200, 44252];
	AX_QTY_MB			: ARRAY[1..3] OF BYTE := [3, 1, 1];
END_VAR
SUPER^.M_StartStop(); 

// Start/Stop
Trig_Local_Start(CLK:=IN_CmdStart_Local);
Trig_Local_Stop(CLK:=IN_CmdStop_Local);

Trig_Start(CLK:=IN_CmdStart);
Trig_Stop(CLK:=IN_CmdStop);

IF Trig_Local_Start.Q OR Trig_Local_Stop.Q OR Trig_Stop.Q OR Trig_Start.Q THEN
	RS_StartStop(SET:=(IN_CmdStart_Local AND NOT IN_CmdStop_Local) OR (IN_CmdStart AND NOT (IN_CmdStop OR IN_CmdStop_Local)), 
			 Reset1 := IN_CmdStop_Local OR (IN_CmdStop AND NOT IN_CmdStart_Local)); 
END_IF

// Emergency stop 
Trig_Local_EmergencyStop(CLK:=IN_CmdEmergencyStop_Local);

// Reset 
Trig_Reset(CLK:= IN_CmdReset_L);

FB_ModbusWrite[5](WriteCmd := FALSE);
FB_ModbusWrite[6](WriteCmd := FALSE);
//FB_ModbusWrite[7](WriteCmd := FALSE);

// Start/Stop/Reset
MesBlockWrite2_Temp[1] := BOOL_TO_WORD(RS_StartStop.Q1);
MesBlockWrite2_Temp[2] := BOOL_TO_WORD(NOT RS_StartStop.Q1);
MesBlockWrite2_Temp[3] := BOOL_TO_WORD(Trig_Reset.Q);
// Emergency stop 
MesBlockWrite3_Temp    			:= BOOL_TO_WORD(Trig_Local_EmergencyStop.Q);

MesDataExd.MesData.OUT_CmdStart := RS_StartStop.Q1 ; 
MesDataExd.MesData.OUT_CmdStop  := NOT RS_StartStop.Q1 ; 	
MesDataExd.OUT_CmdReset			:= 	Trig_Reset.Q;

StartStop_RTrig(CLK:=CalCP_CMD_StartStop);

FB_ModbusWrite[5]
(
	pSrcAddr := ADR (MesBlockWrite2_Temp),
	sIPAddr := ParamIPAddress,
	tTimeout := ParamTimeout,
	nMBAddr := AX_ADR_MB[1],
	nTCPport := ParamTCPPort,
	cbLength := SIZEOF(MesBlockWrite2_Temp),
	nQuantity := AX_QTY_MB[1],
	nUnitID := ParamUnitID,
	WriteCmd := StartStop_RTrig.Q AND MesDataExd.MesData.MesCP_Write ,
	Reset := CmdClearFault_G,
	ErrorId => AX_ModbusWriteAlarmId[5],
	ModbusWriteAlarm => AX_ModbusWriteAlarm[5]
);

	FB_ModbusWrite[6]
(
	pSrcAddr := ADR (MesBlockWrite3_Temp),
	sIPAddr := ParamIPAddress,
	tTimeout := ParamTimeout,
	nMBAddr := AX_ADR_MB[2],
	nTCPport := ParamTCPPort,
	cbLength := SIZEOF(MesBlockWrite3_Temp),
	nQuantity := AX_QTY_MB[2],
	nUnitID := ParamUnitID,
	WriteCmd := Trig_Local_EmergencyStop.Q AND MesDataExd.MesData.MesCP_Write,
	Reset := CmdClearFault_G,
	ErrorId => AX_ModbusWriteAlarmId[6],
	ModbusWriteAlarm => AX_ModbusWriteAlarm[6]
);

// INV watchdog timer: for the first version of the code, this feature is not used and the watchdog is turned timer off. Developped for future uses.
// Write register every second 
//TP_Watchdog(IN:= Watchdog_CP_Write, PT:=TIME#1S);
//FTrig_Watchdog(CLK:=TP_Watchdog.Q);
//Watchdog_CP_Write := FTrig_Watchdog.Q;
//
//MesBlockWrite8_Temp := INT_TO_WORD(1);
//
//	FB_ModbusWrite[7]
//(
//	pSrcAddr  := ADR (MesBlockWrite8_Temp),
//	sIPAddr   := ParamIPAddress,
//	tTimeout  := ParamTimeout,
//	nMBAddr   := AX_ADR_MB[3],
//	nTCPport  := ParamTCPPort,
//	cbLength  := SIZEOF(MesBlockWrite8_Temp),
//	nQuantity := AX_QTY_MB[3],
//	nUnitID   := ParamUnitID,
//	WriteCmd  := MesData.MesCP_Write AND Watchdog_CP_Write,
//	Reset     := CmdClearFault_G,
//	ErrorId => AX_ModbusWriteAlarmId[7],
//	ModbusWriteAlarm => AX_ModbusWriteAlarm[7]
//);
//
END_METHOD

METHOD M_StateManager
//////////////////
// Detect which is the state of the inverter. IF loss of communication MesState =0, the last inverter state is kept  
/////////////////

VAR 
	// Method local variables (reinitialized at each cycle) 

	
END_VAR
//MesState_INV
// 0 = Power Up >3	, 3 = Standby DC>7	, 6 = Ready DC >3	, 9 = Ready>7		, 12 = ON>1		, 15 = Diagnostic AC > 3	
// 1 = Init>3 	, 4 = Precharge DC>3	, 7 = Standby AC>7, 10 = Wait>3 	, 13 = Stop>0 	, 16 = Discharge >5		 			  		
// 2 = OFF>0		, 5 = Softcharge DC >3	, 8 = Blackstart>3, 11 = Pre ON>3	, 14 = Ready AC>3 , 17 = Fault>6

//MesState
//0=Stopped, 1 = MPPT, 2 = Sleeping, 3 = Starting, 4 = Throttled, 5 = Shutting down, 6 = Fault, 7 = Standby

MesDataExd.MesData.MesState := 0; 


IF MesDataExd.MesData.MesState_INV = 13 OR MesDataExd.MesData.MesState_INV = 2 THEN
	MesDataExd.MesData.MesState.0 := 1; 

ELSIF MesDataExd.MesData.MesState_INV = 12 AND MesDataExd.MesStatusCurtail_P.0 THEN
	MesDataExd.MesData.MesState.1 := 1; 
	
ELSIF 	MesDataExd.MesData.MesState_INV = 0 OR MesDataExd.MesData.MesState_INV = 1 OR MesDataExd.MesData.MesState_INV = 4 OR MesDataExd.MesData.MesState_INV = 5 OR 
		MesDataExd.MesData.MesState_INV = 6 OR MesDataExd.MesData.MesState_INV = 8 OR MesDataExd.MesData.MesState_INV = 10 OR MesDataExd.MesData.MesState_INV = 11 OR 
		MesDataExd.MesData.MesState_INV = 14 OR MesDataExd.MesData.MesState_INV = 15 THEN
	MesDataExd.MesData.MesState.3 := 1; 
	
ELSIF MesDataExd.MesData.MesState_INV = 12 AND MesDataExd.MesStatusCurtail_P.2 THEN
	MesDataExd.MesData.MesState.4 := 1;
 
ELSIF MesDataExd.MesData.MesState_INV = 17 THEN
	MesDataExd.MesData.MesState.6 := 1; // Fault 
ELSIF MesDataExd.MesData.MesState_INV = 16 THEN
	MesDataExd.MesData.MesState.5 := 1;  // Discharge
ELSE 
	MesDataExd.MesData.MesState.7 := 1; 
END_IF



SUPER^.M_StateManager();
END_METHOD

END_FUNCTION_BLOCK

// ---- 01_Equipement_Library/Inverter/FB_INV_PE_HEMG3.TcPOU
FUNCTION_BLOCK FB_INV_PE_HEMG3 EXTENDS FB_INV_Base

VAR_INPUT PERSISTENT
		ParamTcpPort				: UINT := 502;					  (* (NA) TCP port *)
		ParamIPAddress				: STRING; 						  (* (NA) Config: IP Adress of PV Inverter *)
		ParamUnitID 				: BYTE; 						  (* (NA) PE SKID Modbus Unit ID *)
		
		ParamSmax					: REAL := 1900;					  (* (kVA) Maximum apparent power of the SKID *)
		ParamID_INV					: UINT := 1;					  (* (NA) INV number 1 or 2 in the SKID *)
		ParamNbDU					: BYTE := 10; 					  (* (NA) Total Number of disconnecting units (cables wired on the PCS) *)				
		ParamNbDU_PowerCol			: ARRAY[1..3] OF BYTE := [5,5,5]; (* (NA) Number of disconnecting uits for each Power Columns *)		
		
		ParamPref_NoCom				: REAL := 100;					  (* (%) P reference defaut value in case Reset refs time different from OFF and loss of communication with PPC *)
		ParamQref_NoCom				: REAL := 0;					  (* (%) Q reference defaut value in case Reset refs time different from OFF and loss of communication with PPC *)
END_VAR

VAR_INPUT 
		IN_CmdEmergencyStop_Local	: BOOL;
		
		IN_SetptQ_Local			: REAL ; 		// (kVar) Local Reactive Power setpoint  
			
		MesDataExd		AT %Q*		: INV_PE_HEMG3; 					   // (NA) Inverter Object 
END_VAR
VAR	
	// M_READ VARIABLES//		
		Trig_Local_EmergencyStop	: R_Trig;
		Trig_Reset					: R_Trig;
		FTrig_Watchdog				: F_Trig;
		Timer_Watchdog				: BOOL;
		Watchdog_CP_Write			: BOOL;
		TP_Watchdog					: TP;
		
